// TwinCAT 3 PLC project PlcPrograme260424
// ProgramVersion: 3.1.4024.0
// libraries:
//   Tc2_EtherCAT, * (Beckhoff Automation GmbH)
//   Tc2_IoFunctions, * (Beckhoff Automation GmbH)
//   Tc2_MC2, * (Beckhoff Automation GmbH)
//   Tc2_ModbusRTU, * (Beckhoff Automation GmbH)
//   Tc2_NC, * (Beckhoff Automation GmbH)
//   Tc2_NcDrive, * (Beckhoff Automation GmbH)
//   Tc2_NCI, * (Beckhoff Automation GmbH)
//   Tc2_PlcInterpolation, * (Beckhoff Automation GmbH)
//   Tc2_SerialCom, * (Beckhoff Automation GmbH)
//   Tc2_Standard, * (Beckhoff Automation GmbH)
//   Tc2_SUPS, * (Beckhoff Automation GmbH)
//   Tc2_System, * (Beckhoff Automation GmbH)
//   Tc2_Utilities, * (Beckhoff Automation GmbH)
//   Tc3_MC2_AdvancedHoming, * (Beckhoff Automation GmbH)
//   Tc3_Module, * (Beckhoff Automation GmbH)
//   Util, * (System)
// project tree:
//   DUTs/Pump/ ST_Pump.TcDUT
//   DUTs/System/ ST_System.TcDUT
//   DUTs/气缸控制/ CylinderStatus.TcDUT, ST_YV.TcDUT
//   DUTs/真空控制/ ST_Vacuum.TcDUT
//   FB/01_Axis/DUTs/Axis_TouchProbeHome/ E_HomeStep.TcDUT, ST_HomeAdsGroup.TcDUT
//   FB/01_Axis/DUTs/Axis_DriveHome/ ST_HomeCoEGroup.TcDUT
//   FB/01_Axis/DUTs/ ST_Axis.TcDUT, ST_AxisControl.TcDUT, ST_AxisParameter.TcDUT, ST_AxisPosControl.TcDUT, ST_AxisPosPar.TcDUT, ST_AxisPosState.TcDUT, ST_AxisPos.TcDUT, ST_AxisState.TcDUT, ST_HomeViaDrivePar.TcDUT
//   FB/01_Axis/FB/ FB_Axis.TcPOU, FB_Axis_PE_Correct.TcPOU, FB_TouchProbe_Home_Bylimit.TcPOU, FB_Drive_Home.TcPOU
//   FB/02_NCI/FB/ FB_013_WriteZeroShiftEx.TcPOU, FB_010_ReadRParameter.TcPOU, FB_011WriteRParameter.TcPOU, FB_012_StepOnAfterStopEx.TcPOU, FB_01_NCI.TcPOU, FB_02_BuidGroup.TcPOU, FB_03_LoadProg.TcPOU, FB_04_Start.TcPOU, FB_05_ClearGrp.TcPOU, FB_06_ExSTOP.TcPOU, FB_07_FastMFunc.TcPOU, FB_08_ReSetEx.TcPOU, FB_09_SetOverridePercent.TcPOU
//   FB/05_YV/ FB_V_3B5.TcPOU
//   FB/06真空控制/ FB_VacuumControl.TcPOU
//   FB/11_AIO/DUTs/ ST_AIO.TcDUT
//   FB/11_AIO/FB/ FB_ADC.TcPOU, FB_DAC.TcPOU
//   FB/31_PDMSCtr/DUTs/ ST_LightCtr.TcDUT
//   FB/31_PDMSCtr/FB/ FB_PDMSCtr.TcPOU
//   FB/02_NCI/DUTs/ ST_IJP.TcDUT
//   FB/51_Netid/ FB_ReadNetid.TcPOU
//   FB/41_PosCom/DUTs/ ST_EL5131_CamCtrl.TcDUT
//   FB/41_PosCom/FB/ FB_013_POS_Comparition.TcPOU
//   FB/61_Alarm/DUTs/ Enum_ErrorClass.TcDUT, ST_Error.TcDUT, ST_HistoryError.TcDUT
//   FB/61_Alarm/FB/ FB_Alarm.TcPOU, FB_SetError.TcPOU, F_FormatWstringErrInfo.TcPOU
//   FB/71_Gear/DOUTs/ ST_Gear.TcDUT
//   FB/71_Gear/FB/ FB_Gear.TcPOU
//   GVLs/ Com_GVLS.TcGVL, GVL_ALM.TcGVL, GVL_IO.TcGVL, Programdata.TcGVL
//   / PlcTask.TcTTO
//   POUs/05_气缸控制/ YV_Ctrl.TcPOU
//   POUs/06_真空控制/ Vac_Ctrl.TcPOU
//   POUs/13_PosCompartion/ POS_Comparition.TcPOU
//   POUs/14_Bump/ Pump.TcPOU
//   POUs/15_Gear/ ProgGear.TcPOU
//   POUs/1_Axis/ AxisLink.TcPOU
//   POUs/2_Nci/ NCI_MAIN.TcPOU
//   POUs/3_Aio/ AIO.TcPOU
//   POUs/07_PDMctr/ PDMctr.TcPOU
//   POUs/ System_State.TcPOU
// real-time tasks:
//   TASK PlcTask: cycle T#1ms, priority 4, ADS port 350
// motion (NC):
//   TASK NC-Task 1 SAF: cycle T#1ms, priority 5, ADS port 501
//   TASK NC-Task 1 SVB: cycle T#2ms, priority 9, ADS port 511
//   AXIS X (id 1)
//     Dynamic: Acceleration=15000, Deceleration=15000, Jerk=150000
//     Velo: RefSync=1, SlowManual=10, FastManual=10, Fast=5
//     OtherSettings: AllowMotionCmdToSlave=true
//     encoder EncType=19
//       EncPara: ScaleFactorNumerator=1, ScaleFactorDenominator=10000, MaxCount=#xffffffff
//     drive DrvType=16
//       DrvPara: MaxCount=#xffffffff, DriveControlDWord=#x00020100
//         Analog: TorqueSetpointScale=10, ScaleFactorActTorque=0.1
//         TimeComp: TaskDelayCycles=1
//     controller CtrType=1
//       CtrPara: PriorControlFactor=1
//         Observer: BandWidth=20
//   AXIS Y (id 2)
//     Dynamic: Acceleration=15000, Deceleration=15000, Jerk=150000
//     Velo: RefSync=1, SlowManual=30, FastManual=30, Fast=5, Maximum=500
//     OtherSettings: AllowMotionCmdToSlave=true
//     encoder EncType=19
//       EncPara: ScaleFactorNumerator=1, ScaleFactorDenominator=10000, MaxCount=#xffffffff
//     drive DrvType=16
//       DrvPara: MaxCount=#xffffffff, DriveControlDWord=#x00020100
//         Analog: VeloReferenz=500, TorqueSetpointScale=10, ScaleFactorActTorque=0.1
//         TimeComp: TaskDelayCycles=1
//     controller CtrType=1
//       CtrPara: PriorControlFactor=1
//         Observer: BandWidth=20
//   AXIS R (id 3)
//     General: UnitName=°
//     Dynamic: AccelerationMaximum=50000, DecelerationMaximum=50000, Acceleration=50000, Deceleration=50000, Jerk=5000000
//     Velo: RefSync=1, SlowManual=5, FastManual=5, Fast=1000
//     OtherSettings: AllowMotionCmdToSlave=true
//     encoder EncType=19
//       EncPara: ScaleFactorNumerator=360, ScaleFactorDenominator=13107200, MaxCount=#xffffffff
//     drive DrvType=16
//       DrvPara: MaxCount=#xffffffff, DriveControlDWord=#x00020100
//         Analog: TorqueSetpointScale=10, ScaleFactorActTorque=0.1
//         TimeComp: TaskDelayCycles=1
//     controller CtrType=1
//       CtrPara: PriorControlFactor=1
//         Observer: BandWidth=20
//   AXIS Z1 (id 4)
//     Velo: RefSync=1, SlowManual=20, FastManual=20, Fast=200
//     OtherSettings: AllowMotionCmdToSlave=true
//     encoder EncType=19
//       EncPara: ScaleFactorNumerator=5, ScaleFactorDenominator=1048576, MaxCount=#xffffffff
//     drive DrvType=16
//       DrvPara: MaxCount=#xffffffff, DriveControlDWord=#x00000100
//         Analog: TorqueSetpointScale=10, ScaleFactorActTorque=0.1
//         TimeComp: TaskDelayCycles=1
//     controller CtrType=1
//       CtrPara: PriorControlFactor=1
//         Observer: BandWidth=20
//   AXIS Z2 (id 5)
//     Velo: RefSync=1, SlowManual=10, FastManual=10, Fast=200
//     OtherSettings: AllowMotionCmdToSlave=true
//     encoder EncType=19
//       EncPara: ScaleFactorNumerator=2, ScaleFactorDenominator=50000, Inverse=true, MaxCount=#xffffffff
//     drive DrvType=16
//       DrvPara: Inverse=true, MaxCount=#xffffffff, DriveControlDWord=#x00020000
//         Analog: TorqueSetpointScale=10, ScaleFactorActTorque=0.1
//         TimeComp: TaskDelayCycles=1
//     controller CtrType=1
//       CtrPara: PriorControlFactor=1
//         Observer: BandWidth=20
//   AXIS Pin (id 6)
//     Dynamic: AccelerationMaximum=5000, DecelerationMaximum=5000, Acceleration=5000, Deceleration=5000, Jerk=50000
//     Velo: SlowManual=3, FastManual=5, Maximum=5500
//     OtherSettings: AllowMotionCmdToSlave=true
//     encoder EncType=19
//       EncPara: ScaleFactorNumerator=360, ScaleFactorDenominator=10000, MaxCount=#xffffffff
//     drive DrvType=16
//       DrvPara: MaxCount=#xffffffff, DriveControlDWord=#x00020000
//         Analog: VeloReferenz=5000, TorqueSetpointScale=10, ScaleFactorActTorque=0.1
//         TimeComp: TaskDelayCycles=1
//     controller CtrType=1
//       CtrPara: PriorControlFactor=1
//         PosDiffControl: Range=50
//         Observer: BandWidth=20
//   AXIS R1 (id 7)
//     Velo: SlowManual=3, FastManual=5
//     OtherSettings: AllowMotionCmdToSlave=true
//     encoder EncType=19
//       EncPara: MaxCount=#xffffffff, ReferenceSystem=1
//     drive DrvType=16
//       DrvPara: MaxCount=#xffffffff, DriveControlDWord=#x00020000
//         Analog: TorqueSetpointScale=10, ScaleFactorActTorque=0.1
//         TimeComp: TaskDelayCycles=1
//     controller CtrType=1
//       CtrPara: PriorControlFactor=1
//         Observer: BandWidth=20
//   AXIS R2 (id 8)
//     Velo: SlowManual=3, FastManual=5
//     OtherSettings: AllowMotionCmdToSlave=true
//     encoder EncType=19
//       EncPara: MaxCount=#xffffffff, ReferenceSystem=1
//     drive DrvType=16
//       DrvPara: MaxCount=#xffffffff, DriveControlDWord=#x00020000
//         Analog: TorqueSetpointScale=10, ScaleFactorActTorque=0.1
//         TimeComp: TaskDelayCycles=1
//     controller CtrType=1
//       CtrPara: PriorControlFactor=1
//         Observer: BandWidth=20
//   AXIS R3 (id 9)
//     Velo: SlowManual=3, FastManual=5
//     OtherSettings: AllowMotionCmdToSlave=true
//     encoder EncType=19
//       EncPara: MaxCount=#xffffffff, ReferenceSystem=1
//     drive DrvType=16
//       DrvPara: MaxCount=#xffffffff, DriveControlDWord=#x00020000
//         Analog: TorqueSetpointScale=10, ScaleFactorActTorque=0.1
//         TimeComp: TaskDelayCycles=1
//     controller CtrType=1
//       CtrPara: PriorControlFactor=1
//         Observer: BandWidth=20
//   AXIS Bump (id 10)
//     Dynamic: Acceleration=100, Deceleration=100, Jerk=500
//     Velo: SlowManual=1, FastManual=3
//     TargetPosControl: Range=0.01
//     OtherSettings: AllowMotionCmdToSlave=true
//     encoder EncType=19
//       EncPara: ScaleFactorNumerator=0.01, ScaleFactorDenominator=10000, MaxCount=#xffffffff
//     drive DrvType=16
//       DrvPara: MaxCount=#xffffffff
//         Analog: TorqueSetpointScale=10, ScaleFactorActTorque=0.1
//         TimeComp: TaskDelayCycles=1
//     controller CtrType=1
//       CtrPara: PriorControlFactor=1
//         PosDiffControl: Enable=false, Range=20
//         Observer: BandWidth=20
// I/O:
//   DEVICE Device 1 (EtherCAT), AmsNetId 192.168.1.50.2.1
//     Term 1 (EK1200) [EK1200-5000 EtherCAT Power supply (2A E-Bus)]
//       Term 2 (EL1889) [EL1889 16Ch. Dig. Input 24V, 3ms, negative]
//       Term 3 (EL1889) [EL1889 16Ch. Dig. Input 24V, 3ms, negative]
//       Term 4 (EL2889) [EL2889 16Ch. Dig. Output 24V, 0.5A, negative]
//       Term 5 (EL3064) [EL3064 4Ch. Ana. Input 0-10V]
//       Term 6 (EL3064) [EL3064 4Ch. Ana. Input 0-10V]
//       Term 7 (EL4004) [EL4004 4Ch. Ana. Output 0-10V, 12bit]
//       Term 8 (EL4004) [EL4004 4Ch. Ana. Output 0-10V, 12bit]
//       Term 11 (EL6002) [EL6002 Interface 2Ch. (RS232)]
//       Term 12 (EK1110) [EK1110 EtherCAT extension]
//     Drive 13 (E2 CoE Drive) [E2 CoE Drive]
//     Drive 14 (E2 CoE Drive) [E2 CoE Drive]
//     Drive 15 (E2 CoE Drive) [E2 CoE Drive]
//     Drive 16 (SGDXS-xxxxA0x CoE Drive) [SGDXS-xxxxA0x EtherCAT(CoE) SERVOPACK Rev02.09]
//     Drive 17 (DM3C-EC522) [DM3C-EC522(COE)]
//     Drive 35 (AZD-KED) [AZD-KED rev0000]
//     Drive 37 (AZD4A-KED-1-3) [AZD4A-KED rev0301]
//     Drive 38 (AZD-KED) [AZD-KED rev0000]
// variable links:
//   NC-Task 1 SAF/Axes/Bump <-> Device 1 (EtherCAT)/Drive 38 (AZD-KED)
//     Drive/Inputs/In/nDcOutputTime <-> InfoData/DcOutputShift
//     Drive/Inputs/In/nState1 <-> Transmit PDO mapping 1/Statusword
//     Drive/Inputs/In/nState2 <-> Transmit PDO mapping 1/Statusword @bit 8
//     Drive/Inputs/In/nState4 @bit 1 <-> WcState/InputToggle
//     Drive/Inputs/In/nState4 <-> WcState/WcState
//     Drive/Inputs/In/nState5 <-> Transmit PDO mapping 1/Modes of operation display
//     Drive/Outputs/Out/nCtrl1 <-> Receive PDO mapping 1/Controlword
//     Drive/Outputs/Out/nCtrl2 <-> Receive PDO mapping 1/Controlword @bit 8
//     Drive/Outputs/Out/nCtrl5 <-> Receive PDO mapping 1/Modes of operation
//     Drive/Outputs/Out/nDataOut1 <-> Receive PDO mapping 1/Target position
//     Enc/Inputs/In/nDataIn1 <-> Transmit PDO mapping 1/Position actual value
//     Enc/Inputs/In/nDcInputTime <-> InfoData/DcInputShift
//     Enc/Inputs/In/nState4 @bit 1 <-> WcState/InputToggle
//     Enc/Inputs/In/nState4 <-> WcState/WcState
//   NC-Task 1 SAF/Axes/Pin <-> Device 1 (EtherCAT)/Drive 35 (AZD-KED)
//     Drive/Inputs/In/nDcOutputTime <-> InfoData/DcOutputShift
//     Drive/Inputs/In/nState1 <-> Transmit PDO mapping 1/Statusword
//     Drive/Inputs/In/nState2 <-> Transmit PDO mapping 1/Statusword @bit 8
//     Drive/Inputs/In/nState4 @bit 1 <-> WcState/InputToggle
//     Drive/Inputs/In/nState4 <-> WcState/WcState
//     Drive/Inputs/In/nState5 <-> Transmit PDO mapping 1/Modes of operation display
//     Drive/Outputs/Out/nCtrl1 <-> Receive PDO mapping 1/Controlword
//     Drive/Outputs/Out/nCtrl2 <-> Receive PDO mapping 1/Controlword @bit 8
//     Drive/Outputs/Out/nCtrl5 <-> Receive PDO mapping 1/Modes of operation
//     Drive/Outputs/Out/nDataOut1 <-> Receive PDO mapping 1/Target position
//     Enc/Inputs/In/nDataIn1 <-> Transmit PDO mapping 1/Position actual value
//     Enc/Inputs/In/nDcInputTime <-> InfoData/DcInputShift
//     Enc/Inputs/In/nState4 @bit 1 <-> WcState/InputToggle
//     Enc/Inputs/In/nState4 <-> WcState/WcState
//   NC-Task 1 SAF/Axes/R <-> Device 1 (EtherCAT)/Drive 15 (E2 CoE Drive)
//     Drive/Inputs/In/nDataIn1 <-> TxPDO 1/Following error actual value
//     Drive/Inputs/In/nDcOutputTime <-> InfoData/DcOutputShift
//     Drive/Inputs/In/nState1 <-> TxPDO 1/Statusword
//     Drive/Inputs/In/nState2 <-> TxPDO 1/Statusword @bit 8
//     Drive/Inputs/In/nState4 @bit 1 <-> WcState/InputToggle
//     Drive/Inputs/In/nState4 <-> WcState/WcState
//     Drive/Inputs/In/nState5 <-> TxPDO 1/Mode of operation display
//     Drive/Outputs/Out/nCtrl1 <-> RxPDO 1/Controlword
//     Drive/Outputs/Out/nCtrl2 <-> RxPDO 1/Controlword @bit 8
//     Drive/Outputs/Out/nCtrl5 <-> RxPDO 1/Mode of operation
//     Drive/Outputs/Out/nDataOut1 <-> RxPDO 1/Target Position
//     Enc/Inputs/In/nDataIn1 <-> TxPDO 1/Position actual value
//     Enc/Inputs/In/nDataIn3 <-> TxPDO 1/Touch Probe 1 positive edge
//     Enc/Inputs/In/nDcInputTime <-> InfoData/DcInputShift
//     Enc/Inputs/In/nState4 @bit 1 <-> WcState/InputToggle
//     Enc/Inputs/In/nState4 <-> WcState/WcState
//     Enc/Inputs/In/nState5 <-> TxPDO 1/Touch Probe status
//     Enc/Inputs/In/nState6 <-> TxPDO 1/Touch Probe status @bit 8
//     Enc/Outputs/Out/nCtrl5 <-> RxPDO 1/Touch probe function
//     Enc/Outputs/Out/nCtrl6 <-> RxPDO 1/Touch probe function @bit 8
//   NC-Task 1 SAF/Axes/R1 <-> Device 1 (EtherCAT)/Drive 37 (AZD4A-KED-1-3)
//     Drive/Inputs/In/nDcOutputTime <-> InfoData/DcOutputShift
//     Drive/Inputs/In/nState1 <-> Axis1 Transmit PDO mapping 1/Statusword
//     Drive/Inputs/In/nState2 <-> Axis1 Transmit PDO mapping 1/Statusword @bit 8
//     Drive/Inputs/In/nState4 @bit 1 <-> WcState/InputToggle
//     Drive/Inputs/In/nState4 <-> WcState/WcState
//     Drive/Inputs/In/nState5 <-> Axis1 Transmit PDO mapping 1/Modes of operation display
//     Drive/Outputs/Out/nCtrl1 <-> Axis1 Receive PDO mapping 1/Controlword
//     Drive/Outputs/Out/nCtrl2 <-> Axis1 Receive PDO mapping 1/Controlword @bit 8
//     Drive/Outputs/Out/nCtrl5 <-> Axis1 Receive PDO mapping 1/Modes of operation
//     Drive/Outputs/Out/nDataOut1 <-> Axis1 Receive PDO mapping 1/Target position
//     Enc/Inputs/In/nDataIn1 <-> Axis1 Transmit PDO mapping 1/Position actual value
//     Enc/Inputs/In/nDcInputTime <-> InfoData/DcInputShift
//     Enc/Inputs/In/nState4 @bit 1 <-> WcState/InputToggle
//     Enc/Inputs/In/nState4 <-> WcState/WcState
//   NC-Task 1 SAF/Axes/R2 <-> Device 1 (EtherCAT)/Drive 37 (AZD4A-KED-1-3)
//     Drive/Inputs/In/nDcOutputTime <-> InfoData/DcOutputShift
//     Drive/Inputs/In/nState1 <-> Axis2 Transmit PDO mapping 1/Statusword
//     Drive/Inputs/In/nState2 <-> Axis2 Transmit PDO mapping 1/Statusword @bit 8
//     Drive/Inputs/In/nState4 @bit 1 <-> WcState/InputToggle
//     Drive/Inputs/In/nState4 <-> WcState/WcState
//     Drive/Inputs/In/nState5 <-> Axis2 Transmit PDO mapping 1/Modes of operation display
//     Drive/Outputs/Out/nCtrl1 <-> Axis2 Receive PDO mapping 1/Controlword
//     Drive/Outputs/Out/nCtrl2 <-> Axis2 Receive PDO mapping 1/Controlword @bit 8
//     Drive/Outputs/Out/nCtrl5 <-> Axis2 Receive PDO mapping 1/Modes of operation
//     Drive/Outputs/Out/nDataOut1 <-> Axis2 Receive PDO mapping 1/Target position
//     Enc/Inputs/In/nDataIn1 <-> Axis2 Transmit PDO mapping 1/Position actual value
//     Enc/Inputs/In/nDcInputTime <-> InfoData/DcInputShift
//     Enc/Inputs/In/nState4 @bit 1 <-> WcState/InputToggle
//     Enc/Inputs/In/nState4 <-> WcState/WcState
//   NC-Task 1 SAF/Axes/R3 <-> Device 1 (EtherCAT)/Drive 37 (AZD4A-KED-1-3)
//     Drive/Inputs/In/nDcOutputTime <-> InfoData/DcOutputShift
//     Drive/Inputs/In/nState1 <-> Axis3 Transmit PDO mapping 1/Statusword
//     Drive/Inputs/In/nState2 <-> Axis3 Transmit PDO mapping 1/Statusword @bit 8
//     Drive/Inputs/In/nState4 @bit 1 <-> WcState/InputToggle
//     Drive/Inputs/In/nState4 <-> WcState/WcState
//     Drive/Inputs/In/nState5 <-> Axis3 Transmit PDO mapping 1/Modes of operation display
//     Drive/Outputs/Out/nCtrl1 <-> Axis3 Receive PDO mapping 1/Controlword
//     Drive/Outputs/Out/nCtrl2 <-> Axis3 Receive PDO mapping 1/Controlword @bit 8
//     Drive/Outputs/Out/nCtrl5 <-> Axis3 Receive PDO mapping 1/Modes of operation
//     Drive/Outputs/Out/nDataOut1 <-> Axis3 Receive PDO mapping 1/Target position
//     Enc/Inputs/In/nDataIn1 <-> Axis3 Transmit PDO mapping 1/Position actual value
//     Enc/Inputs/In/nDcInputTime <-> InfoData/DcInputShift
//     Enc/Inputs/In/nState4 @bit 1 <-> WcState/InputToggle
//     Enc/Inputs/In/nState4 <-> WcState/WcState
//   NC-Task 1 SAF/Axes/X <-> Device 1 (EtherCAT)/Drive 14 (E2 CoE Drive)
//     Drive/Inputs/In/nDataIn1 <-> TxPDO 1/Following error actual value
//     Drive/Inputs/In/nDcOutputTime <-> InfoData/DcOutputShift
//     Drive/Inputs/In/nState1 <-> TxPDO 1/Statusword
//     Drive/Inputs/In/nState2 <-> TxPDO 1/Statusword @bit 8
//     Drive/Inputs/In/nState4 @bit 1 <-> WcState/InputToggle
//     Drive/Inputs/In/nState4 <-> WcState/WcState
//     Drive/Inputs/In/nState5 <-> TxPDO 1/Mode of operation display
//     Drive/Outputs/Out/nCtrl1 <-> RxPDO 1/Controlword
//     Drive/Outputs/Out/nCtrl2 <-> RxPDO 1/Controlword @bit 8
//     Drive/Outputs/Out/nCtrl5 <-> RxPDO 1/Mode of operation
//     Drive/Outputs/Out/nDataOut1 <-> RxPDO 1/Target Position
//     Enc/Inputs/In/nDataIn1 <-> TxPDO 1/Position actual value
//     Enc/Inputs/In/nDataIn3 <-> TxPDO 1/Touch Probe 1 positive edge
//     Enc/Inputs/In/nDcInputTime <-> InfoData/DcInputShift
//     Enc/Inputs/In/nState4 @bit 1 <-> WcState/InputToggle
//     Enc/Inputs/In/nState4 <-> WcState/WcState
//     Enc/Inputs/In/nState5 <-> TxPDO 1/Touch Probe status
//     Enc/Inputs/In/nState6 <-> TxPDO 1/Touch Probe status @bit 8
//     Enc/Outputs/Out/nCtrl5 <-> RxPDO 1/Touch probe function
//     Enc/Outputs/Out/nCtrl6 <-> RxPDO 1/Touch probe function @bit 8
//   NC-Task 1 SAF/Axes/Y <-> Device 1 (EtherCAT)/Drive 13 (E2 CoE Drive)
//     Drive/Inputs/In/nDataIn1 <-> TxPDO 1/Following error actual value
//     Drive/Inputs/In/nDcOutputTime <-> InfoData/DcOutputShift
//     Drive/Inputs/In/nState1 <-> TxPDO 1/Statusword
//     Drive/Inputs/In/nState2 <-> TxPDO 1/Statusword @bit 8
//     Drive/Inputs/In/nState4 @bit 1 <-> WcState/InputToggle
//     Drive/Inputs/In/nState4 <-> WcState/WcState
//     Drive/Inputs/In/nState5 <-> TxPDO 1/Mode of operation display
//     Drive/Outputs/Out/nCtrl1 <-> RxPDO 1/Controlword
//     Drive/Outputs/Out/nCtrl2 <-> RxPDO 1/Controlword @bit 8
//     Drive/Outputs/Out/nCtrl5 <-> RxPDO 1/Mode of operation
//     Drive/Outputs/Out/nDataOut1 <-> RxPDO 1/Target Position
//     Enc/Inputs/In/nDataIn1 <-> TxPDO 1/Position actual value
//     Enc/Inputs/In/nDataIn3 <-> TxPDO 1/Touch Probe 1 positive edge
//     Enc/Inputs/In/nDcInputTime <-> InfoData/DcInputShift
//     Enc/Inputs/In/nState4 @bit 1 <-> WcState/InputToggle
//     Enc/Inputs/In/nState4 <-> WcState/WcState
//     Enc/Inputs/In/nState5 <-> TxPDO 1/Touch Probe status
//     Enc/Inputs/In/nState6 <-> TxPDO 1/Touch Probe status @bit 8
//     Enc/Outputs/Out/nCtrl5 <-> RxPDO 1/Touch probe function
//     Enc/Outputs/Out/nCtrl6 <-> RxPDO 1/Touch probe function @bit 8
//   NC-Task 1 SAF/Axes/Z1 <-> Device 1 (EtherCAT)/Drive 16 (SGDXS-xxxxA0x CoE Drive)
//     Drive/Inputs/In/nDataIn1 <-> 1st Transmit PDO mapping/Following error actual value
//     Drive/Inputs/In/nDataIn3[0] <-> 1st Transmit PDO mapping/Torque actual value
//     Drive/Inputs/In/nDcOutputTime <-> InfoData/DcOutputShift
//     Drive/Inputs/In/nState1 <-> 1st Transmit PDO mapping/Status word
//     Drive/Inputs/In/nState2 <-> 1st Transmit PDO mapping/Status word @bit 8
//     Drive/Inputs/In/nState4 @bit 1 <-> WcState/InputToggle
//     Drive/Inputs/In/nState4 <-> WcState/WcState
//     Drive/Inputs/In/nState5 <-> 1st Transmit PDO mapping/Modes of operation display
//     Drive/Outputs/Out/nCtrl1 <-> 1st Receive PDO mapping/Control word
//     Drive/Outputs/Out/nCtrl2 <-> 1st Receive PDO mapping/Control word @bit 8
//     Drive/Outputs/Out/nCtrl5 <-> 1st Receive PDO mapping/Modes of operation
//     Drive/Outputs/Out/nDataOut1 <-> 1st Receive PDO mapping/Target position
//     Drive/Outputs/Out/nDataOut2 <-> 1st Receive PDO mapping/Target velocity
//     Drive/Outputs/Out/nDataOut4[0] <-> 1st Receive PDO mapping/Target torque
//     Enc/Inputs/In/nDataIn1 <-> 1st Transmit PDO mapping/Position actual value
//     Enc/Inputs/In/nDataIn3 <-> 1st Transmit PDO mapping/Touch probe 1 position value
//     Enc/Inputs/In/nDcInputTime <-> InfoData/DcInputShift
//     Enc/Inputs/In/nState4 @bit 1 <-> WcState/InputToggle
//     Enc/Inputs/In/nState4 <-> WcState/WcState
//     Enc/Inputs/In/nState5 <-> 1st Transmit PDO mapping/Touch probe status
//     Enc/Inputs/In/nState6 <-> 1st Transmit PDO mapping/Touch probe status @bit 8
//     Enc/Outputs/Out/nCtrl5 <-> 1st Receive PDO mapping/Touch probe function
//     Enc/Outputs/Out/nCtrl6 <-> 1st Receive PDO mapping/Touch probe function @bit 8
//   NC-Task 1 SAF/Axes/Z2 <-> Device 1 (EtherCAT)/Drive 17 (DM3C-EC522)
//     Drive/Inputs/In/nDcOutputTime <-> InfoData/DcOutputShift
//     Drive/Inputs/In/nState1 <-> Transmit PDO 1/Status Word
//     Drive/Inputs/In/nState2 <-> Transmit PDO 1/Status Word @bit 8
//     Drive/Inputs/In/nState4 @bit 1 <-> WcState/InputToggle
//     Drive/Inputs/In/nState4 <-> WcState/WcState
//     Drive/Outputs/Out/nCtrl1 <-> Receive PDO 1/Control Word
//     Drive/Outputs/Out/nCtrl2 <-> Receive PDO 1/Control Word @bit 8
//     Drive/Outputs/Out/nDataOut1 <-> Receive PDO 1/Profile Target Position
//     Enc/Inputs/In/nDataIn1 <-> Transmit PDO 1/Position Actual Value
//     Enc/Inputs/In/nDataIn3 <-> Transmit PDO 1/Touch Probe 1 Positive Value
//     Enc/Inputs/In/nDcInputTime <-> InfoData/DcInputShift
//     Enc/Inputs/In/nState4 @bit 1 <-> WcState/InputToggle
//     Enc/Inputs/In/nState4 <-> WcState/WcState
//     Enc/Inputs/In/nState5 <-> Transmit PDO 1/Touch Probe Status
//     Enc/Inputs/In/nState6 <-> Transmit PDO 1/Touch Probe Status @bit 8
//     Enc/Outputs/Out/nCtrl5 <-> Receive PDO 1/Touch Probe Function
//     Enc/Outputs/Out/nCtrl6 <-> Receive PDO 1/Touch Probe Function @bit 8
//   PlcPrograme260424/PlcPrograme260424 Instance <-> Device 1 (EtherCAT)
//     PlcTask Inputs/System_State.fbReadNetid.tAmsNetid <-> InfoData/AmsNetId
//   PlcPrograme260424/PlcPrograme260424 Instance <-> Device 1 (EtherCAT)/Drive 13 (E2 CoE Drive)
//     PlcTask Inputs/Com_GVLS.arstAxis[1].uiSlaveAddr <-> InfoData/AdsAddr/port
//   PlcPrograme260424/PlcPrograme260424 Instance <-> Device 1 (EtherCAT)/Drive 14 (E2 CoE Drive)
//     PlcTask Inputs/Com_GVLS.arstAxis[2].uiSlaveAddr <-> InfoData/AdsAddr/port
//   PlcPrograme260424/PlcPrograme260424 Instance <-> Device 1 (EtherCAT)/Drive 15 (E2 CoE Drive)
//     PlcTask Inputs/Com_GVLS.arstAxis[3].uiSlaveAddr <-> InfoData/AdsAddr/port
//   PlcPrograme260424/PlcPrograme260424 Instance <-> Device 1 (EtherCAT)/Drive 16 (SGDXS-xxxxA0x CoE Drive)
//     PlcTask Inputs/Com_GVLS.arstAxis[4].uiSlaveAddr <-> InfoData/AdsAddr/port
//   PlcPrograme260424/PlcPrograme260424 Instance <-> Device 1 (EtherCAT)/Drive 17 (DM3C-EC522)
//     PlcTask Inputs/Com_GVLS.arstAxis[5].uiSlaveAddr <-> InfoData/AdsAddr/port
//   PlcPrograme260424/PlcPrograme260424 Instance <-> Device 1 (EtherCAT)/Drive 35 (AZD-KED)
//     PlcTask Inputs/Com_GVLS.arstAxis[6].uiSlaveAddr <-> InfoData/AdsAddr/port
//   PlcPrograme260424/PlcPrograme260424 Instance <-> Device 1 (EtherCAT)/Drive 37 (AZD4A-KED-1-3)
//     PlcTask Inputs/Com_GVLS.arstAxis[7].uiSlaveAddr <-> InfoData/AdsAddr/port
//     PlcTask Inputs/Com_GVLS.arstAxis[8].uiSlaveAddr <-> InfoData/AdsAddr/port
//     PlcTask Inputs/Com_GVLS.arstAxis[9].uiSlaveAddr <-> InfoData/AdsAddr/port
//   PlcPrograme260424/PlcPrograme260424 Instance <-> Device 1 (EtherCAT)/Drive 38 (AZD-KED)
//     PlcTask Inputs/Com_GVLS.arstAxis[10].uiSlaveAddr <-> InfoData/AdsAddr/port
//   PlcPrograme260424/PlcPrograme260424 Instance <-> Device 1 (EtherCAT)/Term 1 (EK1200)/Term 11 (EL6002)
//     PlcTask Inputs/PDMctr.FB_PDMSCtr.COMin_MASTER @bit {16..184 step 8} <-> COM TxPDO-Map Inputs Channel 1/Data In {0..21}  (22 links)
//     PlcTask Inputs/PDMctr.FB_PDMSCtr.COMin_MASTER <-> COM TxPDO-Map Inputs Channel 1/Status
//     PlcTask Outputs/PDMctr.FB_PDMSCtr.COMout_MASTER <-> COM RxPDO-Map Outputs Channel 1/Ctrl
//     PlcTask Outputs/PDMctr.FB_PDMSCtr.COMout_MASTER @bit {16..184 step 8} <-> COM RxPDO-Map Outputs Channel 1/Data Out {0..21}  (22 links)
//   PlcPrograme260424/PlcPrograme260424 Instance <-> Device 1 (EtherCAT)/Term 1 (EK1200)/Term 2 (EL1889)
//     PlcTask Inputs/GVL_IO.X000001 <-> Channel 1/Input
//     PlcTask Inputs/GVL_IO.X000002 <-> Channel 2/Input
//     PlcTask Inputs/GVL_IO.X000003 <-> Channel 3/Input
//     PlcTask Inputs/GVL_IO.X000004 <-> Channel 4/Input
//     PlcTask Inputs/GVL_IO.X000005 <-> Channel 5/Input
//     PlcTask Inputs/GVL_IO.X000006 <-> Channel 6/Input
//     PlcTask Inputs/GVL_IO.X000007 <-> Channel 7/Input
//     PlcTask Inputs/GVL_IO.X000008 <-> Channel 8/Input
//     PlcTask Inputs/GVL_IO.X000009 <-> Channel 9/Input
//     PlcTask Inputs/GVL_IO.X000010 <-> Channel 10/Input
//     PlcTask Inputs/GVL_IO.X000011 <-> Channel 11/Input
//     PlcTask Inputs/GVL_IO.X000012 <-> Channel 12/Input
//     PlcTask Inputs/GVL_IO.X000013 <-> Channel 13/Input
//     PlcTask Inputs/GVL_IO.X000014 <-> Channel 14/Input
//     PlcTask Inputs/GVL_IO.X000015 <-> Channel 15/Input
//     PlcTask Inputs/GVL_IO.X000016 <-> Channel 16/Input
//   PlcPrograme260424/PlcPrograme260424 Instance <-> Device 1 (EtherCAT)/Term 1 (EK1200)/Term 3 (EL1889)
//     PlcTask Inputs/GVL_IO.X001001 <-> Channel 1/Input
//     PlcTask Inputs/GVL_IO.X001002 <-> Channel 2/Input
//     PlcTask Inputs/GVL_IO.X001003 <-> Channel 3/Input
//     PlcTask Inputs/GVL_IO.X001004 <-> Channel 4/Input
//     PlcTask Inputs/GVL_IO.X001005 <-> Channel 5/Input
//     PlcTask Inputs/GVL_IO.X001006 <-> Channel 6/Input
//     PlcTask Inputs/GVL_IO.X001007 <-> Channel 7/Input
//     PlcTask Inputs/GVL_IO.X001008 <-> Channel 8/Input
//     PlcTask Inputs/GVL_IO.X001009 <-> Channel 9/Input
//     PlcTask Inputs/GVL_IO.X001010 <-> Channel 10/Input
//     PlcTask Inputs/GVL_IO.X001011 <-> Channel 11/Input
//     PlcTask Inputs/GVL_IO.X001012 <-> Channel 12/Input
//     PlcTask Inputs/GVL_IO.X001013 <-> Channel 13/Input
//     PlcTask Inputs/GVL_IO.X001014 <-> Channel 14/Input
//     PlcTask Inputs/GVL_IO.X001015 <-> Channel 15/Input
//     PlcTask Inputs/GVL_IO.X001016 <-> Channel 16/Input
//   PlcPrograme260424/PlcPrograme260424 Instance <-> Device 1 (EtherCAT)/Term 1 (EK1200)/Term 4 (EL2889)
//     PlcTask Outputs/GVL_IO.Y000001 <-> Channel 1/Output
//     PlcTask Outputs/GVL_IO.Y000002 <-> Channel 2/Output
//     PlcTask Outputs/GVL_IO.Y000003 <-> Channel 3/Output
//     PlcTask Outputs/GVL_IO.Y000004 <-> Channel 4/Output
//     PlcTask Outputs/GVL_IO.Y000005 <-> Channel 5/Output
//     PlcTask Outputs/GVL_IO.Y000006 <-> Channel 6/Output
//     PlcTask Outputs/GVL_IO.Y000007 <-> Channel 7/Output
//     PlcTask Outputs/GVL_IO.Y000008 <-> Channel 8/Output
//     PlcTask Outputs/GVL_IO.Y000009 <-> Channel 9/Output
//     PlcTask Outputs/GVL_IO.Y000010 <-> Channel 10/Output
//     PlcTask Outputs/GVL_IO.Y000011 <-> Channel 11/Output
//     PlcTask Outputs/GVL_IO.Y000012 <-> Channel 12/Output
//     PlcTask Outputs/GVL_IO.Y000013 <-> Channel 13/Output
//     PlcTask Outputs/GVL_IO.Y000014 <-> Channel 14/Output
//     PlcTask Outputs/GVL_IO.Y000015 <-> Channel 15/Output
//     PlcTask Outputs/GVL_IO.Y000016 <-> Channel 16/Output
//   PlcPrograme260424/PlcPrograme260424 Instance <-> Device 1 (EtherCAT)/Term 1 (EK1200)/Term 5 (EL3064)
//     PlcTask Inputs/Programdata.AX_1[{1..4}] <-> AI Standard Channel {1..4}/Value  (4 links)
//   PlcPrograme260424/PlcPrograme260424 Instance <-> Device 1 (EtherCAT)/Term 1 (EK1200)/Term 6 (EL3064)
//     PlcTask Inputs/Programdata.AX_2[{1..4}] <-> AI Standard Channel {1..4}/Value  (4 links)
//   PlcPrograme260424/PlcPrograme260424 Instance <-> Device 1 (EtherCAT)/Term 1 (EK1200)/Term 7 (EL4004)
//     PlcTask Outputs/Programdata.AY_1[{1..4}] <-> AO Outputs Channel {1..4}/Analog output  (4 links)
//   PlcPrograme260424/PlcPrograme260424 Instance <-> Device 1 (EtherCAT)/Term 1 (EK1200)/Term 8 (EL4004)
//     PlcTask Outputs/Programdata.AY_2[{1..4}] <-> AO Outputs Channel {1..4}/Analog output  (4 links)
//   PlcPrograme260424/PlcPrograme260424 Instance <-> NC-Task 1 SAF/Axes/Bump
//     PlcTask Inputs/Programdata.arAXIS[10].NcToPlc <-> Outputs/ToPlc
//     PlcTask Outputs/Programdata.arAXIS[10].PlcToNc <-> Inputs/FromPlc
//   PlcPrograme260424/PlcPrograme260424 Instance <-> NC-Task 1 SAF/Axes/Pin
//     PlcTask Inputs/Programdata.arAXIS[6].NcToPlc <-> Outputs/ToPlc
//     PlcTask Outputs/Programdata.arAXIS[6].PlcToNc <-> Inputs/FromPlc
//   PlcPrograme260424/PlcPrograme260424 Instance <-> NC-Task 1 SAF/Axes/R
//     PlcTask Inputs/Programdata.arAXIS[3].NcToPlc <-> Outputs/ToPlc
//     PlcTask Outputs/Programdata.arAXIS[3].PlcToNc <-> Inputs/FromPlc
//   PlcPrograme260424/PlcPrograme260424 Instance <-> NC-Task 1 SAF/Axes/R1
//     PlcTask Inputs/Programdata.arAXIS[7].NcToPlc <-> Outputs/ToPlc
//     PlcTask Outputs/Programdata.arAXIS[7].PlcToNc <-> Inputs/FromPlc
//   PlcPrograme260424/PlcPrograme260424 Instance <-> NC-Task 1 SAF/Axes/R2
//     PlcTask Inputs/Programdata.arAXIS[8].NcToPlc <-> Outputs/ToPlc
//     PlcTask Outputs/Programdata.arAXIS[8].PlcToNc <-> Inputs/FromPlc
//   PlcPrograme260424/PlcPrograme260424 Instance <-> NC-Task 1 SAF/Axes/R3
//     PlcTask Inputs/Programdata.arAXIS[9].NcToPlc <-> Outputs/ToPlc
//     PlcTask Outputs/Programdata.arAXIS[9].PlcToNc <-> Inputs/FromPlc
//   PlcPrograme260424/PlcPrograme260424 Instance <-> NC-Task 1 SAF/Axes/X
//     PlcTask Inputs/Programdata.arAXIS[1].NcToPlc <-> Outputs/ToPlc
//     PlcTask Outputs/Programdata.arAXIS[1].PlcToNc <-> Inputs/FromPlc
//   PlcPrograme260424/PlcPrograme260424 Instance <-> NC-Task 1 SAF/Axes/Y
//     PlcTask Inputs/Programdata.arAXIS[2].NcToPlc <-> Outputs/ToPlc
//     PlcTask Outputs/Programdata.arAXIS[2].PlcToNc <-> Inputs/FromPlc
//   PlcPrograme260424/PlcPrograme260424 Instance <-> NC-Task 1 SAF/Axes/Z1
//     PlcTask Inputs/Programdata.arAXIS[4].NcToPlc <-> Outputs/ToPlc
//     PlcTask Outputs/Programdata.arAXIS[4].PlcToNc <-> Inputs/FromPlc
//   PlcPrograme260424/PlcPrograme260424 Instance <-> NC-Task 1 SAF/Axes/Z2
//     PlcTask Inputs/Programdata.arAXIS[5].NcToPlc <-> Outputs/ToPlc
//     PlcTask Outputs/Programdata.arAXIS[5].PlcToNc <-> Inputs/FromPlc
//   PlcPrograme260424/PlcPrograme260424 Instance <-> NC-Task 1 SAF/Channel 2
//     PlcTask Inputs/Com_GVLS.stIJP.in_stItpToPlc <-> Outputs/ToPlc
//     PlcTask Outputs/Com_GVLS.stIJP.out_stItpToPlc <-> Inputs/FromPlc

CONFIGURATION PlcPrograme260424
    RESOURCE PLC ON TwinCAT3
        TASK PlcTask(INTERVAL := T#1ms, PRIORITY := 4);
        PROGRAM AxisLink WITH PlcTask : AxisLink;
        PROGRAM NCI_MAIN WITH PlcTask : NCI_MAIN;
        PROGRAM AIO WITH PlcTask : AIO;
        PROGRAM System_State WITH PlcTask : System_State;
        PROGRAM PDMctr WITH PlcTask : PDMctr;
        PROGRAM Vac_Ctrl WITH PlcTask : Vac_Ctrl;
        PROGRAM POS_Comparition WITH PlcTask : POS_Comparition;
        PROGRAM ProgGear WITH PlcTask : ProgGear;
        PROGRAM YV_Ctrl WITH PlcTask : YV_Ctrl;
        PROGRAM Pump WITH PlcTask : Pump;
    END_RESOURCE
END_CONFIGURATION

// ---- DUTs/Pump/ST_Pump.TcDUT
TYPE ST_Pump :
STRUCT
	rJogVel_A								:REAL				    ;			// 流速	
	rJogVol_A								:REAL				    ;			// 容积
	strml               :STRING:='5ml'               ;  //当前进样器容积
	rInjectDia          :ARRAY[1..2] OF REAL  :=[ 7.3, 10.3]; //当前进样器内径
	rVol_Process1   : REAL;  // 流程1：快速注入容量 (ul)
    rVel_Process1   : REAL;  // 流程1：快速注入流速 (ul/min)
    rVel_Process2   : REAL;  // 流程2：匀速注入流速 (ul/min)
    rVol_Process3   : REAL;  // 流程3：快速抽取容量 (ul)
    rVel_Process3   : REAL;  // 流程3：快速抽取流速 (ul/min)
	iCurrentStep    : INT;    // 当前运行状态 (0:待机, 10:注入准备, 11:快速注入中..., 20:匀速注入中..., 30:抽取中..., 31:抽取中...)
	bEX_PumpTrigOn  : BOOL;   //注射泵触发开
	bEX_PumpTrigOff  : BOOL;   //注射泵触发关

END_STRUCT
END_TYPE

// ---- DUTs/System/ST_System.TcDUT
TYPE ST_System :
STRUCT
	    strNetID                                                               :STRING;
        bSystemPowerOn                                        :BOOL                                                        ;                        //系统动力电上电标志        
        bManual                                                        :BOOL                                                        ;                        //手自动标志
        bReset                                                        :BOOL                                                        ;                        //复位
        bStop                                                        :BOOL                                                        ;                        //停止
        bEMG                                                               :BOOL                                                        ;                        //急停
        bSafetyDoor                                                :BOOL                                                        ;                        //安全门
        bLightOn                                                :BOOL                                                        ;                        //照明灯
        bAxesPowerOK                                            :BOOL                                                        ;                        //所有轴均上使能
        bAxesHomeOK                                                :BOOL                                                        ;                        //所有轴均回零完成
	bHOME                             :BOOL                                      ;           // 整机回零
	bHoming                           :BOOL                                      ;           // 整机回零中
	bHOMEOK                           :BOOL                                      ;           // 整机回零完成
	bPower                            :BOOL                                      ;           // 整机使能
	bPowerOK                          :BOOL                                      ;           // 整机使能完成
	bUVon                             :BOOL                                      ;           // UV开关
	bUVErr                            :BOOL                                      ;           // UV开关报错
        bAxesInMotion                                        :BOOL                                                        ;                        //有轴移动
        bError                                                        :BOOL                                                        ;                        //报错
        bWarning                                                :BOOL                                                        ;                        //警告
        bLightError                                                :BOOL                                                        ;                        //轻量错误
        bCriticalError                                        :BOOL                                                        ;                        //严重错误
        bErrorUpdate                                        :BOOL                                                           ;                        //出现新的报错                                        
        arErrorID                                                :ARRAY[0..999] OF BOOL                                     ;                        //报警索引号
        arstrErrorInfo                                        :ARRAY[0..999] OF STRING                                      ;                        //报警信息（英）
        strDeviceName                                        :STRING                                                        ;                        //设备名称
        uiPinNum                                                :UINT                                                        ;                        //剥离头类型，1-单电机，2-双电机
	    bSignalLampRed	                                       :BOOL	; // 三色灯-红                   
        bSignalLampGreen	                                    :BOOL	 ;// 三色灯-绿
        bSignalLampYellow	                                     :BOOL	 ;// 三色灯-黄
        bSingalLampBuzzle	                                      :BOOL	; // 三色灯-蜂鸣器
END_STRUCT
END_TYPE

// ---- DUTs/气缸控制/CylinderStatus.TcDUT
(* 单个气缸状态 *)
TYPE CylinderStatus :
STRUCT
    bExtendReq    : BOOL;   // 伸出请求
    bRetractReq   : BOOL;   // 回缩请求
    q_bExtend     : BOOL;   // 输出伸出
    q_bRetract    : BOOL;   // 输出回缩
    xExtendPos    : BOOL;   // 伸出到位
    xRetractPos   : BOOL;   // 回缩到位
    bInDeadtime   : BOOL;   // 死区标志
    bAlarm        : BOOL;   // 报警状态
END_STRUCT
END_TYPE

// ---- DUTs/气缸控制/ST_YV.TcDUT
TYPE ST_YV :
STRUCT
	bYVFw_A   :BOOL; //  伸出操作
	bYVBw_A   :BOOL; //  缩回操作
	bYVFw_In  :BOOL; //  伸出限位
	bYVBw_In  :BOOL; //  缩回限位
	bYVFw_OK  :BOOL; //  气缸伸出到位
	bYVBw_OK  :BOOL; //  气缸缩回到位
	bYVFw_Out :BOOL; //  硬件输出
	bYVBw_Out :BOOL; //  硬件输出
	bError	  :BOOL; //  错误状态
	//arErrorID :UINT; //  错误ID
	udiError  :UDINT; //  错误ID
	arErrorID	  :ARRAY[0..7] OF BOOL   ;   // 错误ID,上位机需求

END_STRUCT
END_TYPE

// ---- DUTs/真空控制/ST_Vacuum.TcDUT
(*

TYPE ST_Vacuum :
STRUCT
    (* 输入 *)
    bVacuumReq     : BOOL;   // 抽真空请求
    bReleaseReq    : BOOL;   // 破真空请求
    xVacuumOk      : BOOL;   // 真空到位信号

    (* 输出 *)
    qVacuumValve   : BOOL;   // 真空阀
    qReleaseValve  : BOOL;   // 破真空阀

    (* 状态 *)
    bVacuumDone    : BOOL;
    bAlarm         : BOOL;
END_STRUCT
END_TYPE

*)

TYPE ST_Vacuum :
STRUCT
    (* 输入 *)
    bVacuumReq      : BOOL;   // 抽真空请求
END_STRUCT
END_TYPE

// ---- FB/01_Axis/DUTs/Axis_TouchProbeHome/E_HomeStep.TcDUT
//{attribute 'qualified_only'}
{attribute 'strict'}
TYPE E_HomeStep :
(
	IndexHomeInital:=0,
	AckHomeDirection,
	SetParameter,
	SetParameterState,
	ReadParameter,
	ReadParameterState,
	AckParameter,
	ExecuteToOrigin,
	HomeMonitorState,
	HomeMoveABS,
	ExecuteHomeDone,
	IndexHomeErrorState
);
END_TYPE

// ---- FB/01_Axis/DUTs/Axis_TouchProbeHome/ST_HomeAdsGroup.TcDUT
TYPE ST_HomeAdsGroup :
STRUCT
    nCalibrationVel			:UDINT:=16#4001;				(* 回零速度ADS地址*)	
	nHomeInfo				:UDINT:=16#5001;				(* 回零参数ADS地址*)

END_STRUCT
END_TYPE

// ---- FB/01_Axis/DUTs/Axis_DriveHome/ST_HomeCoEGroup.TcDUT
TYPE ST_HomeCoEGroup :
STRUCT
	strNetID			    :STRING:='192.168.1.50.2.1';				(* 回零速度coe地址*)	
	wSlaveAddr				:WORD:=1001;				                (* 回零参数coe地址*)
	uiAxisChannelNum        :WORD:=1;                                   (* 一拖多驱动器COE地址递增index*)
END_STRUCT
END_TYPE

// ---- FB/01_Axis/DUTs/ST_Axis.TcDUT
TYPE ST_Axis :
STRUCT
	strName			:STRING					    ;
	wstrName		:WSTRING				    ;
	strNetID        :STRING;
	uiSlaveAddr     AT%I*  :WORD;
	Control			:ST_AxisControl				;		
	Parameter		:ST_AxisParameter			;		
	State			:ST_AxisState				;	
	Pos				:ST_AxisPos		            ;
END_STRUCT
END_TYPE

// ---- FB/01_Axis/DUTs/ST_AxisControl.TcDUT

TYPE ST_AxisControl :
STRUCT
	bPowerOn			:BOOL				;		//伺服使能	
	bHome_M				:BOOL				;		//手动回零	
	bHome_A				:BOOL				;		//自动回零	
	bHome_Con			:BOOL				;		//回零条件	
	bJogCw_M			:BOOL				;		//手动点动加（顺时针）	
	bJogCcw_M			:BOOL				;		//手动点动减（逆时针）	
	bJogCw_A			:BOOL				;		//自动点动加（顺时针）	
	bJogCcw_A			:BOOL				;		//自动点动减（逆时针）		
	bJogCw_Con			:BOOL				;		//点动加条件	
	bJogCcw_Con			:BOOL				;		//点动减条件	
	bStop_A				:BOOL				;		//自动停止	
	bStop_M				:BOOL				;		//手动停止	
	bSetPos				:BOOL				;		//置位	
	iJogMode			:INT				;		//Jog运行模式0-连续 1-点动
	bReset_A			:BOOL				;
	bReset_M			:BOOL				;
END_STRUCT
END_TYPE

// ---- FB/01_Axis/DUTs/ST_AxisParameter.TcDUT
TYPE ST_AxisParameter :
STRUCT	
	rMaxVel									:REAL				;			//额定最大速度	
	rHmOffset								:REAL				;			//原点偏差值(单原点回零时使用)	
	rHmVel									:REAL				;			//回零速度	
	rHmAcc									:REAL				;			//回零加速度	
	rHmDec									:REAL				;			//回零减速度	
	rHmJerk									:REAL				;			//回零跃度	
	rJogVel_M								:REAL				;			//手动点动速度	
	rJogAcc_M								:REAL				;			//手动点动加速度	
	rJogDec_M								:REAL				;			//手动点动减速度
	rJogPos_M								:REAL				;			//手动寸动增量	
	rJogVel_A								:REAL				;			//自动点动速度	
	rJogAcc_A								:REAL				;			//自动点动加速度	
	rJogDec_A								:REAL				;			//自动点动减速度	
	rJogPos_A								:REAL				;			//自动寸动增量	
	rStopDec								:REAL				;			//停止减速度	
	rStopJerk								:REAL				;			//停止跃度	
	rSetPos									:REAL				;			//置位位置	
	udiPDO_60FD				AT%I*			:UDINT				;			//限位原点接入驱动器下配置：数字输入
	udiPDO_6071				AT%Q*			:INT				;			// 输入力矩
//	uiPDO_60B8				AT%Q*			:UINT				;			//探针回零模式下配置：探针控制字
//	uiPDO_60B9				AT%I*			:UINT				;			//探针回零模式下配置：探针状态字	
	uiHomeMode								:UINT				;			//0=碰限位回零 , 1=单原点回零 , 2=限位+原点光电回零,6=驱动器回零,8=模块限位+驱动器回零	
	iTorque									:INT				;			//设定转矩
	bAbsEnc									:BOOL				;			//true= 绝对值编码器，false= 增量式编码器	
	bHmDir									:BOOL				;			//FALSE=正向回零 , TRUE=反向回零	
//	diPDO_60BA		 		AT%I*			:DINT				;			//探针回零模式下配置：探针1上升沿	
	diPDO_6064								:DINT				;			//轴当前脉冲数
	rInPosValue                     		:REAL	:=0.01		;			// 运动到位
	rSetPosition							:REAL				;			// 回退距离
	uiAxisChannelNum						:UINT	:=1			;			//针对多轴驱动器中的轴通道号,单轴按通道1计算
	rTorque                                 :REAL               ;           // 力矩模式设定力矩6071
	sthomeViaDrivePar 				:ST_HomeViaDrivePar			;			
END_STRUCT
END_TYPE

// ---- FB/01_Axis/DUTs/ST_AxisPosControl.TcDUT
TYPE ST_AxisPosControl :
STRUCT
	bGo_Con			:			BOOL			;		//定位条件
	bGo_M			:			BOOL			;		//手动定位启动
	bGo_A			:			BOOL			;		//自动定位启动
END_STRUCT
END_TYPE

// ---- FB/01_Axis/DUTs/ST_AxisPosPar.TcDUT
TYPE ST_AxisPosPar :
STRUCT
	bRelEnable			:BOOL		;		//FALSE绝对定位，TRUE相对定位	
	rPos				:REAL		;		//定位位置	
	rVel				:REAL		;		//定位速度	
	rAcc				:REAL		;		//定位加速度	
	rDec				:REAL		;		//定位减速度	
	rJerk				:REAL		;		//定位跃度	
END_STRUCT
END_TYPE

// ---- FB/01_Axis/DUTs/ST_AxisPosState.TcDUT
TYPE ST_AxisPosState :
STRUCT
	bGo_OK			:BOOL		;		//定位完成	
	bGo_Moving		:BOOL		;		//定位中	
	rGo_CT			:REAL		;		//定位持续时间	
END_STRUCT
END_TYPE

// ---- FB/01_Axis/DUTs/ST_AxisPos.TcDUT
TYPE ST_AxisPos :
STRUCT
	Ctrl			:			ST_AxisPosControl	;
	Par				:			ST_AxisPosPar		;
	State			:			ST_AxisPosState		;
END_STRUCT
END_TYPE

// ---- FB/01_Axis/DUTs/ST_AxisState.TcDUT
TYPE ST_AxisState :
STRUCT
	uiNodeAddr									:UINT									;			//从站节点地址		
	rActModuloPos								:REAL									;			//实际位置-模轴位置
	rActPos										:REAL									;			//实际位置-线性位置
	rActVel										:REAL									;			//实际速度	
	rActAcc										:REAL									;			//实际加速度	
	rActTrq										:REAL									;			//实际扭矩	
	bDirPositive								:BOOL									;			//正向运动标志	
	bDirNegative								:BOOL									;			//负向运动标志	
	bPowerOK									:BOOL									;			//使能完成	
	bHoming										:BOOL									;			//回零中	
	bHome_OK									:BOOL									;			//回零完成	
	siModeOfOperation						    :SINT					                ;		    //  驱动器输出PLC工作模式，传递给PLC的工作模式	
	bPSw										:BOOL									;			//正极限	
	bNSw										:BOOL									;			//负极限	
	bHSw										:BOOL									;			//原点开关	
	bStandStill									:BOOL									;			//停止中
	bMoving										:BOOL									;			//移动中
	bHasJob                                     :BOOL									;			//工作中
	bInSync										:BOOL									;			//耦合中	
	bError										:BOOL									;			//报错
	bWarning									:BOOL									;			//警告
	bLightEror									:BOOL									;			//轻量错误
	bCriticalError								:BOOL									;			//严重错误
	arErrorID									:ARRAY[1..12] OF BOOL					;			//错误ID
	udiNCErrorID								:UDINT									;			//NC ErrorID
	uiDriveErrorCode							:UINT									;			//驱动器报警代码
END_STRUCT	
END_TYPE

// ---- FB/01_Axis/DUTs/ST_HomeViaDrivePar.TcDUT
TYPE ST_HomeViaDrivePar :
STRUCT
	//必须设定的参数
//	nCtrl1					AT%I*			:				USINT					;				// 驱动器回零模式下配置 : NC输出的控制字1，传递给PLC 
//	nCtrl2					AT%I*			:				USINT					;				// 驱动器回零模式下配置 : NC输出的控制字1，传递给PLC 
//	ControlWord				AT%Q*			:				UINT					;				// 驱动器回零模式下配置 : PLC输出控制字，传递给驱动器的控制字 
	ModeOfOperation			AT%Q*			:				SINT					;				// 驱动器回零模式下配置 : PLC输出驱动器工作模式，传递给驱动器的工作模式		
	//根据驱动器的实际需求进行设置
	siHomeMethod							:				SINT					;				// 设置通过驱动器回零的方式
	udiHomeVelHigh							:				UDINT					;				// 设置通过驱动器回零的高速回零速度
	udiHomeVelLow							:				UDINT					;				// 设置通过驱动器回零的低速回零速度
	udiHomeAcc								:				UDINT					;				// 设置通过驱动器回零的加减速度
	diHomeOffset							:				DINT					;				// 设置通过驱动器回零的回零偏置
	rHomeVelHigh							:				LREAL					;				// 设置通过探针回零的高速回零速度
	rHomeVelLow							    :				LREAL					;				// 设置通过探针回零的低速回零速度
	rHomeOffset							    :				LREAL					;				// 设置通过探针回零的回零偏置
END_STRUCT
END_TYPE

// ---- FB/11_AIO/DUTs/ST_AIO.TcDUT
TYPE ST_AIO :
STRUCT
	rAI1				:			REAL			;			// 底部负压表显示
	rAI2				:			REAL			;			// 针头气压表显示
	rAI3				:			REAL			;			// 
	rAI4				:			REAL			;			// 
	rAI5				:			REAL			;			// 底部负压比例阀反馈
	rAI6				:			REAL			;			// 针头负压比例阀反馈
	rAI7				:			REAL			;			// 针头正压比例阀反馈
	rAI8				:			REAL			;			//
	rAI9				:			REAL			;			//
	rAI10				:			REAL			;			//
	rAI11				:			REAL			;			//
	rAI12				:			REAL			;			//
	rAI13				:			REAL			;			//
	rAI14				:			REAL			;			//
	rAI15				:			REAL			;			//
	rAI16				:			REAL			;			//
	rAI17				:			REAL			;			//
	rAI18				:			REAL			;			//
	rAI19				:			REAL			;			//
	rAI20				:			REAL			;			//

	rAO1				:			REAL			;			// 底部负压比例阀设定
	rAO2				:			REAL			;			// 针头负压比例阀设定
	rAO3				:			REAL			;			// 针头正压比例阀设定
	rAO4				:			REAL			;			//
	rAO5				:			REAL			;			//
	rAO6				:			REAL			;			//
	rAO7				:			REAL			;			//
	rAO8				:			REAL			;			//
	rAO9				:			REAL			;			//
	rAO10				:			REAL			;			//
	rAO11				:			REAL			;			//
	rAO12				:			REAL			;			//
	rAO13				:			REAL			;			//
	rAO14				:			REAL			;			//
	rAO15				:			REAL			;			//
	rAO16				:			REAL			;			//
END_STRUCT
END_TYPE

// ---- FB/31_PDMSCtr/DUTs/ST_LightCtr.TcDUT
TYPE ST_LightCtr :
STRUCT
	iChannel1ValueSet		:				UINT						;			//通道1设定值
	iChannel2ValueSet		:				UINT						;			//通道2设定值
	iChannel3ValueSet		:				UINT						;			//通道3设定值
	iChannel4ValueSet		:				UINT						;			//通道4设定值
	iChannel1ActValue		:				UINT						;			//通道1当前值
	iChannel2ActValue		:				UINT						;			//通道2当前值
	iChannel3ActValue		:				UINT						;			//通道3当前值
	iChannel4ActValue		:				UINT						;			//通道4当前值
END_STRUCT
END_TYPE

// ---- FB/02_NCI/DUTs/ST_IJP.TcDUT
TYPE ST_IJP :
STRUCT
	in_stItpToPlc AT %I*: NCTOPLC_NCICHANNEL_REF;
	out_stItpToPlc AT %Q*:  PLCTONC_NCICHANNEL_REF;
	strNciName			    :STRING(255)			    ;           // NCI通道名
	bBuildGroupExe			:BOOL				        ;			// 将NC轴添加进NCI通道中 —— 触发
	bClearGroupExe			:BOOL				        ;			// 清除NCI通道中的轴，释放轴 —— 触发
	bLoadPGMExe			    :BOOL				        ;			// G代码装载
	bStartExe			    :BOOL				        ;			// 启动NC通道
	bStopExe			    :BOOL				        ;			// 停止NC通道
	bEstopExe			    :BOOL				        ;			// 紧急停止NCI
	bItpEStopEx             : BOOL ;                                 //  暂停G代码
	bItpStepOnAfterEStopEx  : BOOL                    ;               //  继续G代码
	bAfterEstopExe			:BOOL				        ;			// 紧急停止后恢复
	bResetExe			    :BOOL				        ;			// 错误复位
	bWriteRParExe			:BOOL				        ;				// 写R变量
	bReadRParExe			:BOOL				        ;				// 读R变量
	bLayerChanging			:BOOL				        ;				// 图层切换标志
	bLayerChanged			:BOOL				        ;	       // 图层切换指令
	bPrintDone			    :BOOL				        ;           // 轨迹执行完成
	bLoadPGMDone			:BOOL				        ;    // load路径文件完成
	bEx_TrigH			    :BOOL				        ;		    // 高压触发	输出到硬件
    bEx_Trig			        :BOOL				        ;		    // 阀触发	输出到硬件	
	bEx_TrigHfb			              :BOOL				        ;		    // 手动高压触发	输出到硬件反馈
    bEx_Trigfb			              :BOOL				        ;		    // 手动阀触发	输出到硬件反馈	
    EL5131_CamCtrlMax       :int                        ;// 最大位置比较数组量	
	arrWriteRPar			:ARRAY[0..19] OF LREAL		;
	arrReadRPar			    :ARRAY[0..19] OF LREAL		;
    bEx_TrigEl5131          :BOOL				        ;		    // 位置比较触发允许		
    bWriteZeroShiftExe      :BOOL;
	bEx_TrigBumpBack		:BOOL;								//开泵回抽模式
	lZeroShiftX             :LREAL                      ;           //X偏移值
	lZeroShiftY             :LREAL                      ;           //Y偏移值
	lZeroShiftZ             :LREAL                      ;           //Z偏移值


	

    rPosTolerance           :LREAL :=0.01                     ;           //位置比较允许误差
	tEndPosDelay            :TIME   :=T#1S                       ;           //终点比较延迟时间
//	bTrigSwitch             :BOOL                       ;           //位置比较高压是否开启(on=开)
//	bTrigPreSwitch          :BOOL                       ;          //比置比较例阀是否开启(on=开)
		
    bEl5131_TrigH:  BOOL;                                         //  (1-X1/Y1/Z1位置触发) (2-X1/Y2/Z1位置触发) (3-X2/Y1/Z2位置触发) (4-X2/Y2/Z2位置触发)
    bEl5131_Trig :  BOOL;
 
	strPRGName			    :STRING(255)			    ;           // 文件名
	lrOverrideSet			:LREAL				        ;			// 速度比例设定
	iJetOnDelay			    :INT:=1						;			// 喷墨开延时
	iJetOffDelay			:INT						;			// 喷墨关延时

//	udiErrOutToPlc                  AT%I*                     :UDINT;            // NCI故障码
//    lrPathVeloOutToPlc              AT%I*                     :LREAL ;           // NCI合成速度
	arErrorID									:ARRAY[1..7] OF BOOL;			//错误ID
	udiError									:UDINT			    ;// 错误编号
	bError										:BOOL													;			// 错误标志
    bErrorEStop                                  : BOOL ;                    ;            //  G代码暂停错误标志
	
END_STRUCT
END_TYPE

// ---- FB/41_PosCom/DUTs/ST_EL5131_CamCtrl.TcDUT
TYPE ST_EL5131_CamCtrl :
STRUCT
    // ------------------- 输入变量（控制指令） -------------------
	rPosStart1				 :	LREAL;// 比较起点位置x
	rPosStart2				 :	LREAL;// 比较起点位置y
	rPosStart3				 :	LREAL;// 比较起点位置z
	rPosEnd1                 :	LREAL;// 比较终点位置x
	rPosEnd2                 :	LREAL;// 比较终点位置y
	rPosEnd3                 :	LREAL;// 比较终点位置z
	bCamCtrlStartEn                 :	BOOL;// 比较点执行许可标志
	bCamCtrlEndEn                   :	BOOL;// 比较点执行许可标志
	udiAxisId1               :UDINT                      ;           // 参与位置比较轴ID
	udiAxisId2               :UDINT                      ;           // 参与位置比较轴ID
	udiAxisId3               :UDINT                      ;           // 参与位置比较轴ID
END_STRUCT
END_TYPE

// ---- FB/61_Alarm/DUTs/Enum_ErrorClass.TcDUT
TYPE Enum_ErrorClass :
(
    NoAlarm                		:=0,					//无警报
    Message      				:=1,					//信息
    Event           			:=2,					//事件
    Reserve3		            :=3,					//预留
    Reserve4                   	:=4,					//预留
    Reserve5                   	:=5,					//预留
    LightError          		:=6,					//轻微报警
    CriticalError               :=7						//重度报警
);
END_TYPE

// ---- FB/61_Alarm/DUTs/ST_Error.TcDUT
TYPE ST_Error :
STRUCT
    (*InPut*)
	iErrorID					:					INT						;			//报警ID号
    wstrErrorMessage			:					WSTRING					;			//报警信息
    dtErrorOccorTime			:                   DT						;			//报警发生时间
	bErrorExe					:					BOOL					;			//报警触发信号接入
	bFilterOn					:					BOOL					;			//输入信号滤波功能
	timeFilter					:                   TIME					;			//滤波时间设定
	bResetSignalUse				:					BOOL					;			//启用复位信号复位.true=复位信号为1时且触发信号为0时，复位报警状态;  false=仅触发信号为0时复位报警信号
	bResetExe					:					BOOL					;			//报警复位信号接入
	enumErrorClass				:					Enum_ErrorClass			;			//报警等级

	bAlarmAction1				:					BOOL					;			//报警后输出动作1
	bAlarmAction2				:					BOOL					;			//报警后输出动作2
	bAlarmAction3				:					BOOL					;			//报警后输出动作3
	bAlarmAction4				:					BOOL					;			//报警后输出动作4

   (*OutPut*)
	bErrorOccur					:					BOOL					;			//报警正在发生
	bEnabled					:                	BOOL					;			//当前报警已启用
END_STRUCT
END_TYPE;

// ---- FB/61_Alarm/DUTs/ST_HistoryError.TcDUT
TYPE ST_HistoryError :
STRUCT
  	wstrErrorMessage				:            	WSTRING					;	//报警信息
	iErrorID						:				INT						;	//报警ID号
   	dtErrorTime						:               DT						;	//报警发生时间
END_STRUCT
END_TYPE

// ---- FB/71_Gear/DOUTs/ST_Gear.TcDUT
TYPE ST_Gear :
STRUCT
	wstrName		           :WSTRING	;
    AxisRefMaster  				: Axis_Ref;
	AxisRefSlave   				: Axis_Ref;			        
	bGearIn                     :BOOL;         // 耦合变量
	bFlyGearIn                  :BOOL;         //  飞剪耦合变量
	bGearOut                    :BOOL;         // 耦合变量
	bStop_A                     :BOOL;        //  运动停止
	rRatioNumerator           :LREAL;         // 从轴速度
	uiRatioDenominator        :UINT;         // 主轴速度
	bInSyncing                :BOOL;         // 耦合中
	bFlyInSyncing                :BOOL;         // 耦合中
	bnoInSyncing                 :BOOL;         // 解耦
	rMasterSyncPosition      :LREAL;         // 主轴同步位置
	rSlaveSyncPosition       :LREAL;         // 从轴同步位置
	rSyncVelocity            :LREAL;         // 同步最大速度
	rSyncACC                 :LREAL;
	rSyncDEC                 :LREAL;
	rSyncJerk                :LREAL;
	bError	                 :BOOL;          //  错误状态
	arErrorID				 :ARRAY[1..3] OF BOOL;			//错误ID
END_STRUCT
END_TYPE

// ---- GVLs/Com_GVLS.TcGVL

VAR_GLOBAL
   (* 结构体申明*)
   stSystem          : ST_System:=(strDeviceName:='EHD');
   arstAxis            : ARRAY[1..10] OF ST_Axis;  
   stIJP             : ST_IJP     := (strNciName:='C:\NC\1.nc',lrOverrideSet := LREAL#100);   
   stAIO             : ST_AIO;   
   stLightCtr        : ST_LightCtr;
   arstCamCtrlIO       : ARRAY[1..100] OF ST_EL5131_CamCtrl; //1-X轴 2-Y轴
   bPlatformVacON    :BOOL       :=FALSE;(*真空吸附*)
   bPlatformVacOff   :BOOL       :=FALSE;
   arstHomeADS          :ARRAY[1..10] OF ST_HomeAdsGroup;
   arstHomeCoE          :ARRAY[1..10] OF ST_HomeCoEGroup;
   arstYV					: ARRAY[1..15] OF ST_YV; //所有气缸定义   
   arstVac				:ARRAY[1..15] OF ST_Vacuum; //所有真空定义
   stPump				:ST_Pump;
   arstGear           :ARRAY[1..2] OF ST_Gear;
END_VAR

// ---- GVLs/GVL_ALM.TcGVL
VAR_GLOBAL
	//当前正在发生的警报数量
	iActErrorNum					:             		INT																;
	//历史发生的警报数量
	iHistoryErrorNum				:           		INT																;
	//报警信息数组，根据iErrorIDMax设定上限值。根据需求扩展。
	arrstError						:					ARRAY [1..iErrorIDMax] OF ST_Error								;
	//当前正在发生的报警存储数组，预设30组数据
	arrstActError					:					ARRAY [1..30] OF ST_HistoryError								;
	//清除历史报警信息数组触发变量
	bClearHistoryError				:            		BOOL															;
	//获取的当前系统时间，配合报警信息输出
	tActSystemTime					: 					TIMESTRUCT														;
	// 报警信息中英文选择，默认为中文
	bLanguageSet					:					BOOL															;
END_VAR
VAR_GLOBAL PERSISTENT
	//历史报警存储数组，预设200组数组
	arrstHistoryError				:					ARRAY [1..200] OF ST_HistoryError								;			
END_VAR
VAR_GLOBAL CONSTANT
	// 报警数组最大值，根据实际需求更改
	iErrorIDMax: INT := 500;
END_VAR
VAR_GLOBAL
	bGetSystemTimeDone: BOOL;
END_VAR

// ---- GVLs/GVL_IO.TcGVL
VAR_GLOBAL
(*X*)
	X000001  AT%I*:  BOOL;   // 急停
	X000002  AT%I*:  BOOL;   // X- NO
	X000003  AT%I*:  BOOL;   // x+ NO
	X000004  AT%I*:  BOOL;   // Y- NO
	X000005  AT%I*:  BOOL;   // y+ NO
	X000006  AT%I*:  BOOL;   // 
	X000007  AT%I*:  BOOL;   // 
	X000008  AT%I*:  BOOL;   // Z1+NC 
	X000009  AT%I*:  BOOL;   // Z1-NC 
	X000010  AT%I*:  BOOL;   // Z2+NC 
	X000011  AT%I*:  BOOL;   // Z2-NC 
	X000012  AT%I*:  BOOL;   // 
	X000013  AT%I*:  BOOL;   // 
	X000014  AT%I*:  BOOL;   // 
	X000015  AT%I*:  BOOL;   // 
	X000016  AT%I*:  BOOL;   // 
	
	X001001  AT%I*:  BOOL;   // R1+ 
	X001002  AT%I*:  BOOL;   // R1-
	X001003  AT%I*:  BOOL;   // R2+
	X001004  AT%I*:  BOOL;   // R2-
	X001005  AT%I*:  BOOL;   // R3+
	X001006  AT%I*:  BOOL;   // R3-
	X001007  AT%I*:  BOOL;   // BUMP+
	X001008  AT%I*:  BOOL;   // bump-
	X001009  AT%I*:  BOOL;   // 
	X001010  AT%I*:  BOOL;   // 
	X001011  AT%I*:  BOOL;   // 
	X001012  AT%I*:  BOOL;   // 
	X001013  AT%I*:  BOOL;   // 
	X001014  AT%I*:  BOOL;   // 
	X001015  AT%I*:  BOOL;   // 
	X001016  AT%I*:  BOOL;   // 
	
(*Y*)	
	Y000001 AT%Q*:  BOOL;   // 针头正负压切换阀
	Y000002 AT%Q*:  BOOL;   // 
	Y000003 AT%Q*:  BOOL;   // 
	Y000004 AT%Q*:  BOOL;   // 气缸开
	Y000005 AT%Q*:  BOOL;   //	气缸关 
	Y000006 AT%Q*:  BOOL;   // 	真空破1
	Y000007 AT%Q*:  BOOL;   //  真空吸1
	Y000008 AT%Q*:  BOOL;   //  真空破2
	Y000009 AT%Q*:  BOOL;   //  真空吸2
	Y000010 AT%Q*:  BOOL;   //  真空吸3
	Y000011 AT%Q*:  BOOL;   //  真空破3
	Y000012 AT%Q*:  BOOL;   // 
	Y000013 AT%Q*:  BOOL;   // 
	Y000014 AT%Q*:  BOOL;   // 
	Y000015 AT%Q*:  BOOL;   // 
	Y000016 AT%Q*:  BOOL;   // 高压输出
END_VAR

// ---- GVLs/Programdata.TcGVL
VAR_GLOBAL
	(* *******PTP/NCI*********** *)
	arAXIS:ARRAY[1..10] OF AXIS_REF;
	
	tonSystemFirstRun:TON;
	posEdgeFirstRun:R_TRIG;
	//in_stItpToPlc AT %I*:NCTOPLC_NCICHANNEL_REF;
	//out_stItpToPlc AT %Q*:PLCTONC_NCICHANNEL_REF;
	
	(* ******AIO****** *)	
	AX_1 AT%I*: ARRAY[1..4]  OF INT;// 根据3064、3062、3061情况确定数组长度
	AX_2 AT%I*: ARRAY[1..4]  OF INT;
	AY_1 AT%Q*: ARRAY[1..4]  OF INT;// 根据4004、4002情况确定数组长度
	AY_2 AT%Q*: ARRAY[1..4]  OF INT;

	(**************************************************************************)
	// stXDescPitch: ST_CompensationDesc := (fPosMin:=0.0, fPosMax:=100.0, nTableElements:=11)---安捷伦激光干涉仪补偿表取反,单位mm;
   stXPitchTable: ARRAY[0..20] OF ST_CompensationElement :=[(fPos:=0.0, fCompensation:=0.0),
                                                           (fPos:=10.0, fCompensation:=0.0),
                                                           (fPos:=20.0, fCompensation:=0.0),
                                                           (fPos:=30.0, fCompensation:=0.0),
                                                           (fPos:=40.0, fCompensation:=0.0),
                                                           (fPos:=50.0, fCompensation:=0.0),
                                                           (fPos:=60.0, fCompensation:=0.0),
                                                           (fPos:=70.0, fCompensation:=0.0),
                                                           (fPos:=80.0, fCompensation:=0.0),
                                                           (fPos:=90.0, fCompensation:=0.0),
                                                           (fPos:=100.0, fCompensation:=0.0),
                                                           (fPos:=110.0, fCompensation:=0.0),
                                                           (fPos:=120.0, fCompensation:=0.0),
                                                           (fPos:=130.0, fCompensation:=0.0),
                                                           (fPos:=140.0, fCompensation:=0.0),
                                                           (fPos:=150.0, fCompensation:=0.0),
                                                           (fPos:=160.0, fCompensation:=0.0),
                                                           (fPos:=170.0, fCompensation:=0.0),
                                                           (fPos:=180.0, fCompensation:=0.0),
                                                           (fPos:=190.0, fCompensation:=0.0),
                                                           (fPos:=200.0, fCompensation:=0.0)];
   //stYDescPitch: ST_CompensationDesc := (fPosMin:=0.0, fPosMax:=100.0, nTableElements:=11)---安捷伦激光干涉仪补偿表取反,单位mm;
   stYPitchTable: ARRAY[0..15] OF ST_CompensationElement :=[(fPos:=0.0, fCompensation:=0),
                                                           (fPos:=10.0, fCompensation:=-0.0),
                                                           (fPos:=20.0, fCompensation:=-0.0),
                                                           (fPos:=30.0, fCompensation:=-0.0),
                                                           (fPos:=40.0, fCompensation:=-0.0),
                                                           (fPos:=50.0, fCompensation:=-0.0),
                                                           (fPos:=60.0, fCompensation:=-0.0),
                                                           (fPos:=70.0, fCompensation:=-0.0),
                                                           (fPos:=80.0, fCompensation:=-0.0),
                                                           (fPos:=90.0, fCompensation:=-0.0),
                                                           (fPos:=100.0, fCompensation:=-0.0),
                                                           (fPos:=110.0, fCompensation:=-0.0),
                                                           (fPos:=120.0, fCompensation:=-0.0),
                                                           (fPos:=130.0, fCompensation:=-0.0),
                                                           (fPos:=140.0, fCompensation:=-0.0),
                                                           (fPos:=150.0, fCompensation:=-0.0)];
	(**************************************************************************) 
    
    (**)  
    bXProhibitFwMvALM		:			BOOL:=TRUE			;		(*	X 正向运动禁止报警*)
	bXProhibitBwMvALM		:			BOOL:=TRUE			;		(*	X 负向运动禁止报警*)
	
    bYProhibitFwMvALM		:			BOOL:=TRUE			;		(*	Y 正向运动禁止报警*)
	bYProhibitBwMvALM		:			BOOL:=TRUE			;		(*	Y 负向运动禁止报警*)
	
	bRProhibitFwMvALM		:			BOOL:=TRUE			;		(*	R 正向运动禁止报警*)
	bRProhibitBwMvALM		:			BOOL:=TRUE			;		(*	R 负向运动禁止报警*)
	
	bZ1ProhibitFwMvALM		:			BOOL:=TRUE			;		(*	Z1 正向运动禁止报警*)
	bZ1ProhibitBwMvALM		:			BOOL:=TRUE			;		(*	Z1 负向运动禁止报警*)
	
	bZ2ProhibitFwMvALM		:			BOOL:=TRUE			;		(*	Z2 正向运动禁止报警*)
	bZ2ProhibitBwMvALM		:			BOOL:=TRUE			;		(*	Z2 负向运动禁止报警*)
	
    (*从站号*)
    uiSlaveNum: UINT;
END_VAR

// ---- POUs/1_Axis/AxisLink.TcPOU
PROGRAM AxisLink
VAR
	fbAxis    :ARRAY[1..10] OF FB_Axis;//根据轴数量定义数组
	bFirstRun :BOOL;                  //上电初始化轴参数
	i         :INT;                   //用于轴报错
	fbAxisPECorect:ARRAY[1..2] OF FB_Axis_PE_Correct;
END_VAR

(*****************************************************************
1.轴PROG程序进行默认参数初始化并进行块调用及转system报错ID

2.	bPowerOn		     	// 伺服使能，置1操作,无自复位
    bHome_A				    // 回零,置1操作,无自复位
	bJogCw_A		        // 连续运动正向,上升沿作用,无自复位
	bJogCcw_A			    // 连续运动负向,上升沿作用,无自复位		
	bRelMove_A              // 相对移动,,上升沿作用,无自复位	
	bAbsMove_A              // 绝对移动,上升沿作用,无自复位	
	bStop_A				    // 自动停止,上升沿作用,自复位			
	bHomeStop               // 回零停止,上升沿作用,自复位	
	bReset_A			    // 复位,上升沿作用,自复位
	
3.	nCtrl1                  // link NC参数 --驱动回零轴，NC和驱动controlword通过程序关联 }
	nCtrl2                  // link NC参数 --驱动回零轴，NC和驱动controlword通过程序关联 }--控制字回零用
	ControlWord             // link PDO -- 6040,控制字                                   }
	ModeOfOperation         // link PDO -- 6060,模式切换
	iTorque                 // 设定扭矩 -- 6071,设定扭矩 

4.  uiMaxTorque 			// 最大扭矩     6072   onlineCOE,单位%
 	udiMaxVel 			    // 最大扭矩     607F   onlineCOE,单位P
 	HomeMethod              // 回零方法     6098   onlineCOE
    HomeOffset              // 回零偏置     607C   onlineCOE,单位P
 	HomSwitchVelo           // 驱动寻Z速度  6099.2 onlineCOE,单位P
  
5.	ModeOfOperationdis      // Readcoe-- 6061,控制模式反馈
	ActTorque 			    // Readcoe--6077 读取驱动器实际力矩 
	ErrorCode               // Readcoe-- 603F读取驱动器错误码   
	StatusWord              // Readcoe-- 6041 回零程序中驱动器状态字
	
6.  探针回零不使用上述2-5项配置
*****************************************************************)
(* 参数初始化*)
posEdgeFirstRun(CLK:=NOT bFirstRun);
IF posEdgeFirstRun.Q AND bFirstRun  =FALSE THEN;
arstAxis[1].Parameter.bAbsEnc:=FALSE;
arstAxis[1].Parameter.uiHomeMode:=8;
arstAxis[1].Parameter.bHmDir:=TRUE;
arstAxis[1].Parameter.sthomeViaDrivePar.diHomeOffset:=0;
//arstAxis[1].Parameter.sthomeViaDrivePar.siHomeMethod:=34;
arstAxis[1].Parameter.sthomeViaDrivePar.udiHomeVelHigh:=10;
arstAxis[1].Parameter.sthomeViaDrivePar.udiHomeVelLow:=5;
arstAxis[1].Parameter.sthomeViaDrivePar.udiHomeAcc:=3000;
arstAxis[1].Control.bHome_Con:=TRUE;
arstAxis[1].Parameter.rHmVel:=20;
arstAxis[1].Parameter.rJogVel_A:=100;
arstAxis[1].Parameter.rJogAcc_A:=3000;
arstAxis[1].Parameter.rJogDec_A:=3000;
arstAxis[1].Parameter.rStopDec:=30000;
arstAxis[1].Parameter.rStopJerk:=arstAxis[1].Parameter.rStopDec*50;
arstAxis[1].Parameter.sthomeViaDrivePar.ModeOfOperation:=8;
arstAxis[1].Control.bJogCw_Con:=TRUE;
arstAxis[1].Control.bJogCcw_Con:=TRUE;
arstAxis[1].Pos.Ctrl.bGo_Con:=TRUE;
arstAxis[1].Parameter.rInPosValue:=0.01;  // 到位阈值
arstAxis[1].Parameter.sthomeViaDrivePar.rHomeOffset:=0.0;
arstAxis[1].Parameter.sthomeViaDrivePar.rHomeVelHigh:=10.0;
arstAxis[1].Parameter.sthomeViaDrivePar.rHomeVelLow:=5.0;

arstAxis[2].Parameter.bAbsEnc:=FALSE;
arstAxis[2].Parameter.uiHomeMode:=8;
arstAxis[2].Parameter.bHmDir:=TRUE;
arstAxis[2].Parameter.sthomeViaDrivePar.diHomeOffset:=0;
//arstAxis[2].Parameter.sthomeViaDrivePar.siHomeMethod:=34;
arstAxis[2].Parameter.sthomeViaDrivePar.udiHomeVelHigh:=10;
arstAxis[2].Parameter.sthomeViaDrivePar.udiHomeVelLow:=5;
arstAxis[2].Parameter.sthomeViaDrivePar.udiHomeAcc:=3000;
arstAxis[2].Control.bHome_Con:=TRUE;
arstAxis[2].Parameter.rHmVel:=20;
arstAxis[2].Parameter.rJogVel_A:=100;
arstAxis[2].Parameter.rJogAcc_A:=3000;
arstAxis[2].Parameter.rJogDec_A:=3000;
arstAxis[2].Parameter.rStopDec:=30000;
arstAxis[2].Parameter.rStopJerk:=arstAxis[2].Parameter.rStopDec*10;
arstAxis[2].Parameter.sthomeViaDrivePar.ModeOfOperation:=8;
arstAxis[2].Control.bJogCw_Con:=TRUE;
arstAxis[2].Control.bJogCcw_Con:=TRUE;
arstAxis[2].Pos.Ctrl.bGo_Con:=TRUE;
arstAxis[2].Parameter.rInPosValue:=0.01;  // 到位阈值
arstAxis[2].Parameter.sthomeViaDrivePar.rHomeOffset:=0.0;
arstAxis[2].Parameter.sthomeViaDrivePar.rHomeVelHigh:=10.0;
arstAxis[2].Parameter.sthomeViaDrivePar.rHomeVelLow:=5.0;

arstAxis[3].Parameter.bAbsEnc:=FALSE;
arstAxis[3].Parameter.uiHomeMode:=0;
arstAxis[3].Parameter.bHmDir:=TRUE;
arstAxis[3].Control.bHome_Con:=TRUE;
arstAxis[3].Parameter.rHmVel:=20;
arstAxis[3].Parameter.rJogVel_A:=30;
arstAxis[3].Parameter.rJogAcc_A:=300;
arstAxis[3].Parameter.rJogDec_A:=300;
arstAxis[3].Parameter.rStopDec:=20000;
arstAxis[3].Parameter.rStopJerk:=arstAxis[3].Parameter.rStopDec*20;
arstAxis[3].Parameter.sthomeViaDrivePar.ModeOfOperation:=8;
arstAxis[3].Control.bJogCw_Con:=TRUE;
arstAxis[3].Control.bJogCcw_Con:=TRUE;
arstAxis[3].Pos.Ctrl.bGo_Con:=TRUE;
arstAxis[3].Parameter.sthomeViaDrivePar.rHomeOffset:=0.0;
arstAxis[3].Parameter.sthomeViaDrivePar.rHomeVelHigh:=2.0;
arstAxis[3].Parameter.sthomeViaDrivePar.rHomeVelLow:=1.0;

arstAxis[4].Parameter.bAbsEnc:=FALSE;
arstAxis[4].Parameter.uiHomeMode:=0;
arstAxis[4].Parameter.bHmDir:=TRUE;
arstAxis[4].Control.bHome_Con:=TRUE;
arstAxis[4].Parameter.rHmVel:=20;
arstAxis[4].Parameter.rJogVel_A:=30;
arstAxis[4].Parameter.rJogAcc_A:=300;
arstAxis[4].Parameter.rJogDec_A:=300;
arstAxis[4].Parameter.rStopDec:=20000;
arstAxis[4].Parameter.rStopJerk:=arstAxis[3].Parameter.rStopDec*20;
arstAxis[4].Parameter.sthomeViaDrivePar.ModeOfOperation:=8;
arstAxis[4].Control.bJogCw_Con:=TRUE;
arstAxis[4].Control.bJogCcw_Con:=TRUE;
arstAxis[4].Pos.Ctrl.bGo_Con:=TRUE;
arstAxis[4].Parameter.sthomeViaDrivePar.rHomeOffset:=0.0;
arstAxis[4].Parameter.sthomeViaDrivePar.rHomeVelHigh:=2.0;
arstAxis[4].Parameter.sthomeViaDrivePar.rHomeVelLow:=1.0;

arstAxis[5].Parameter.bAbsEnc:=FALSE;
arstAxis[5].Parameter.uiHomeMode:=0;
arstAxis[5].Parameter.bHmDir:=TRUE;
arstAxis[5].Control.bHome_Con:=TRUE;
arstAxis[5].Parameter.rHmVel:=20;
arstAxis[5].Parameter.rJogVel_A:=30;
arstAxis[5].Parameter.rJogAcc_A:=300;
arstAxis[5].Parameter.rJogDec_A:=300;
arstAxis[5].Parameter.rStopDec:=20000;
arstAxis[5].Parameter.rStopJerk:=arstAxis[3].Parameter.rStopDec*20;
arstAxis[5].Parameter.sthomeViaDrivePar.ModeOfOperation:=8;
arstAxis[5].Control.bJogCw_Con:=TRUE;
arstAxis[5].Control.bJogCcw_Con:=TRUE;
arstAxis[5].Pos.Ctrl.bGo_Con:=TRUE;
arstAxis[5].Parameter.sthomeViaDrivePar.rHomeOffset:=0.0;
arstAxis[5].Parameter.sthomeViaDrivePar.rHomeVelHigh:=2.0;
arstAxis[5].Parameter.sthomeViaDrivePar.rHomeVelLow:=1.0;

arstAxis[6].Parameter.bAbsEnc:=TRUE;
arstAxis[6].Parameter.uiHomeMode:=0;
arstAxis[6].Parameter.bHmDir:=TRUE;
arstAxis[6].Control.bHome_Con:=TRUE;
arstAxis[6].Parameter.rHmVel:=20;
arstAxis[6].Parameter.rJogVel_A:=30;
arstAxis[6].Parameter.rJogAcc_A:=300;
arstAxis[6].Parameter.rJogDec_A:=300;
arstAxis[6].Parameter.rStopDec:=20000;
arstAxis[6].Parameter.rStopJerk:=arstAxis[3].Parameter.rStopDec*20;
arstAxis[6].Parameter.sthomeViaDrivePar.ModeOfOperation:=8;
arstAxis[6].Control.bJogCw_Con:=TRUE;
arstAxis[6].Control.bJogCcw_Con:=TRUE;
arstAxis[6].Pos.Ctrl.bGo_Con:=TRUE;
arstAxis[6].Parameter.sthomeViaDrivePar.rHomeOffset:=0.0;
arstAxis[6].Parameter.sthomeViaDrivePar.rHomeVelHigh:=2.0;
arstAxis[6].Parameter.sthomeViaDrivePar.rHomeVelLow:=1.0;

arstAxis[7].Parameter.bAbsEnc:=FALSE;
arstAxis[7].Parameter.uiHomeMode:=0;
arstAxis[7].Parameter.bHmDir:=TRUE;
arstAxis[7].Control.bHome_Con:=TRUE;
arstAxis[7].Parameter.rHmVel:=20;
arstAxis[7].Parameter.rJogVel_A:=30;
arstAxis[7].Parameter.rJogAcc_A:=300;
arstAxis[7].Parameter.rJogDec_A:=300;
arstAxis[7].Parameter.rStopDec:=20000;
arstAxis[7].Parameter.rStopJerk:=arstAxis[3].Parameter.rStopDec*20;
arstAxis[7].Parameter.sthomeViaDrivePar.ModeOfOperation:=8;
arstAxis[7].Control.bJogCw_Con:=TRUE;
arstAxis[7].Control.bJogCcw_Con:=TRUE;
arstAxis[7].Pos.Ctrl.bGo_Con:=TRUE;
arstAxis[7].Parameter.sthomeViaDrivePar.rHomeOffset:=0.0;
arstAxis[7].Parameter.sthomeViaDrivePar.rHomeVelHigh:=2.0;
arstAxis[7].Parameter.sthomeViaDrivePar.rHomeVelLow:=1.0;
arstAxis[7].Parameter.uiAxisChannelNum:=1;


arstAxis[8].Parameter.bAbsEnc:=FALSE;
arstAxis[8].Parameter.uiHomeMode:=0;
arstAxis[8].Parameter.bHmDir:=TRUE;
arstAxis[8].Control.bHome_Con:=TRUE;
arstAxis[8].Parameter.rHmVel:=20;
arstAxis[8].Parameter.rJogVel_A:=30;
arstAxis[8].Parameter.rJogAcc_A:=300;
arstAxis[8].Parameter.rJogDec_A:=300;
arstAxis[8].Parameter.rStopDec:=20000;
arstAxis[8].Parameter.rStopJerk:=arstAxis[3].Parameter.rStopDec*20;
arstAxis[8].Parameter.sthomeViaDrivePar.ModeOfOperation:=8;
arstAxis[8].Control.bJogCw_Con:=TRUE;
arstAxis[8].Control.bJogCcw_Con:=TRUE;
arstAxis[8].Pos.Ctrl.bGo_Con:=TRUE;
arstAxis[8].Parameter.sthomeViaDrivePar.rHomeOffset:=0.0;
arstAxis[8].Parameter.sthomeViaDrivePar.rHomeVelHigh:=2.0;
arstAxis[8].Parameter.sthomeViaDrivePar.rHomeVelLow:=1.0;
arstAxis[8].Parameter.uiAxisChannelNum:=2;

arstAxis[9].Parameter.bAbsEnc:=FALSE;                                        
arstAxis[9].Parameter.uiHomeMode:=0;                                         
arstAxis[9].Parameter.bHmDir:=TRUE;                                          
arstAxis[9].Control.bHome_Con:=TRUE;                                         
arstAxis[9].Parameter.rHmVel:=20;                                            
arstAxis[9].Parameter.rJogVel_A:=30;                                         
arstAxis[9].Parameter.rJogAcc_A:=300;                                        
arstAxis[9].Parameter.rJogDec_A:=300;                                        
arstAxis[9].Parameter.rStopDec:=20000;                                        
arstAxis[9].Parameter.rStopJerk:=arstAxis[3].Parameter.rStopDec*20;          
arstAxis[9].Parameter.sthomeViaDrivePar.ModeOfOperation:=8;                  
arstAxis[9].Control.bJogCw_Con:=TRUE;                                        
arstAxis[9].Control.bJogCcw_Con:=TRUE;                                       
arstAxis[9].Pos.Ctrl.bGo_Con:=TRUE;                                          
arstAxis[9].Parameter.sthomeViaDrivePar.rHomeOffset:=0.0;                    
arstAxis[9].Parameter.sthomeViaDrivePar.rHomeVelHigh:=2.0;                   
arstAxis[9].Parameter.sthomeViaDrivePar.rHomeVelLow:=1.0;                    
arstAxis[9].Parameter.uiAxisChannelNum:=3;

arstAxis[10].Parameter.bAbsEnc:=FALSE;                                       
arstAxis[10].Parameter.uiHomeMode:=0;                                        
arstAxis[10].Parameter.bHmDir:=TRUE;                                         
arstAxis[10].Control.bHome_Con:=TRUE;                                        
arstAxis[10].Parameter.rHmVel:=1;                                           
arstAxis[10].Parameter.rJogVel_A:=1;                                        
arstAxis[10].Parameter.rJogAcc_A:=10;                                       
arstAxis[10].Parameter.rJogDec_A:=10;                                       
arstAxis[10].Parameter.rStopDec:=100;                                       
arstAxis[10].Parameter.rStopJerk:=arstAxis[3].Parameter.rStopDec*20;         
arstAxis[10].Parameter.sthomeViaDrivePar.ModeOfOperation:=8;                 
arstAxis[10].Control.bJogCw_Con:=TRUE;                                       
arstAxis[10].Control.bJogCcw_Con:=TRUE;                                      
arstAxis[10].Pos.Ctrl.bGo_Con:=TRUE;                                         
arstAxis[10].Parameter.sthomeViaDrivePar.rHomeOffset:=0.0;                   
arstAxis[10].Parameter.sthomeViaDrivePar.rHomeVelHigh:=1.0;                  
arstAxis[10].Parameter.sthomeViaDrivePar.rHomeVelLow:=1.0;                   

// 轴parameter地址
arstHomeADS[1].nCalibrationVel:=16#4001;
arstHomeADS[1].nHomeInfo:=16#5001;
arstHomeADS[2].nCalibrationVel:=16#4002;
arstHomeADS[2].nHomeInfo:=16#5002;
arstHomeADS[3].nCalibrationVel:=16#4003;
arstHomeADS[3].nHomeInfo:=16#5003;
arstHomeADS[4].nCalibrationVel:=16#4004;
arstHomeADS[4].nHomeInfo:=16#5004;
arstHomeADS[5].nCalibrationVel:=16#4005;
arstHomeADS[5].nHomeInfo:=16#5005;
arstHomeADS[6].nCalibrationVel:=16#4006;
arstHomeADS[6].nHomeInfo:=16#5006;

arstHomeADS[7].nCalibrationVel:=16#4007;
arstHomeADS[7].nHomeInfo:=16#5007;

arstHomeADS[8].nCalibrationVel:=16#4008;
arstHomeADS[8].nHomeInfo:=16#5008;

arstHomeADS[9].nCalibrationVel:=16#4009;
arstHomeADS[9].nHomeInfo:=16#5009;

arstHomeADS[10].nCalibrationVel:=16#400A;
arstHomeADS[10].nHomeInfo:=16#500A;

bFirstRun             :=TRUE;
END_IF
(* 轴块调用*)
A_01_AX();
A_02_AY();
A_03_AR();
A_04_AZ1();
A_05_AZ2();
A_06_APin();
A_07_R1();
A_08_R2();
A_09_R3();
A_10_Bump();
(* 轴补偿调用*)
fbAxisPECorect[1](
	AxisRef:= arAXIS[1], 
	arstPitchTable:= stXPitchTable, 
	bEnable:= , 
	bAxisHomeOK:= arstAxis[1].State.bHome_OK, 
	bBacklashDir:= , 
	rBcaklash:= , 
	rDistance:= 0, 
	lrCurBacklash=> , 
	lrCOmpensation=> , 
	bBusy=> , 
	bError=> );
(* 轴补偿调用*)
fbAxisPECorect[2](
	AxisRef:= arAXIS[2], 
	arstPitchTable:= stYPitchTable, 
	bEnable:= , 
	bAxisHomeOK:= arstAxis[2].State.bHome_OK, 
	bBacklashDir:= , 
	rBcaklash:= , 
	rDistance:= 0, 
	lrCurBacklash=> , 
	lrCOmpensation=> , 
	bBusy=> , 
	bError=> );

ACTION A_01_AX:
//Axis-BasicParameterSettings
// 限位默认常闭，常开需要取反,白色常开/黑色常闭
// 轴基础参数设定
arstAxis[1].wstrName:=" 喷涂X轴" ;
arstAxis[1].strNetID:=stSystem.strNetID;//'192.168.1.50.2.1';//arAXIS[1].DriveAddress.NetID;
//arstAxis[1].uiSlaveAddr; 通过drive-infoData-AMSNETID-PORT关联;
arstAxis[1].State.bNSw:= NOT  X000002 ;// PM-l25倍福接黑线，pmac接黑线 
arstAxis[1].State.bPSw:= NOT  X000003 ;


// 力矩
//stAxis[1].Parameter.uiMaxTorque:=800;
// 功能块
fbAxis[1](AxisRef:=arAXIS[1] , stAxis:=arstAxis[1] ,stHomeADS:=arstHomeADS[1], stHomeCoe:=arstHomeCoE[1],stSystem:=stSystem );
END_ACTION

ACTION A_02_AY:
//Axis-BasicParameterSettings
//限位默认常闭，常开需要取反,白色常闭/黑色常开
arstAxis[2].wstrName:=" 喷涂Y轴" ;
arstAxis[2].strNetID:=stSystem.strNetID;///'192.168.1.50.2.1';
//stAxis[2].Parameter.uiSlaveAddr:=1012;通过drive-infoData-AMSNETID-PORT关联;
arstAxis[2].State.bNSw:=NOT X000004 ;// NC-White
arstAxis[2].State.bPSw:=NOT X000005 ;//
//false=etercat
// 功能块
fbAxis[2](AxisRef:=arAXIS[2] , stAxis:=arstAxis[2] , stSystem:=stSystem , stHomeCoe:=arstHomeCoE[1],stHomeADS:=arstHomeADS[2]);
END_ACTION

ACTION A_03_AR:
//Axis-BasicParameterSettings
//限位默认常闭，常开需要取反,白色常闭/黑色常开
arstAxis[3].wstrName:=" 喷涂R轴" ;
arstAxis[3].strNetID:=stSystem.strNetID;//'192.168.1.50.2.1';
//arstAxis[3].Parameter.uiSlaveAddr:=1014;通过drive-infoData-AMSNETID-PORT关联;
arstAxis[3].State.bNSw:= X000014 ;// NC-White
//stAxis[3].State.bHSW:= X000013;
arstAxis[3].State.bPSw:= X000013 ;//
//false=etercat
// 功能块
fbAxis[3](AxisRef:=arAXIS[3] , stAxis:=arstAxis[3] , stSystem:=stSystem  , stHomeCoe:=arstHomeCoE[1],stHomeADS:=arstHomeADS[3]);
END_ACTION

ACTION A_04_AZ1:
//Axis-BasicParameterSettings
//限位默认常闭，常开需要取反,白色常闭/黑色常开
arstAxis[4].wstrName:=" 喷涂Z1轴" ;
arstAxis[4].strNetID:=stSystem.strNetID;//'192.168.1.50.2.1';
//arstAxis[4].Parameter.uiSlaveAddr:=1015;通过drive-infoData-AMSNETID-PORT关联;
arstAxis[4].State.bNSw:= X000009 ;// NC-White
arstAxis[4].State.bPSw:= X000008 ;//
//false=etercat
// 功能块
fbAxis[4](AxisRef:=arAXIS[4] , stAxis:=arstAxis[4] , stSystem:=stSystem  , stHomeCoe:=arstHomeCoE[1],stHomeADS:=arstHomeADS[4]);
END_ACTION

ACTION A_05_AZ2:
//Axis-BasicParameterSettings
//限位默认常闭，常开需要取反,白色常闭/黑色常开
arstAxis[5].wstrName:=" 喷涂Z2轴" ;
arstAxis[5].strNetID:=stSystem.strNetID;//'192.168.1.50.2.1';
//arstAxis[5].Parameter.uiSlaveAddr:=1016;通过drive-infoData-AMSNETID-PORT关联;
arstAxis[5].State.bNSw:= X000011 ;// NC-White
arstAxis[5].State.bPSw:= X000010 ;//
//false=etercat
// 功能块
fbAxis[5](AxisRef:=arAXIS[5] , stAxis:=arstAxis[5] , stSystem:=stSystem , stHomeCoe:=arstHomeCoE[1],stHomeADS:=arstHomeADS[5]);
END_ACTION

ACTION A_06_APin:
//Axis-BasicParameterSettings
//限位默认常闭，常开需要取反,白色常闭/黑色常开
arstAxis[6].wstrName:=" 顶pin轴" ;
arstAxis[6].strNetID:=stSystem.strNetID;//'192.168.1.50.2.1';
//arstAxis[6].Parameter.uiSlaveAddr:=1017;
arstAxis[6].State.bNSw:= TRUE ;// NC-White
arstAxis[6].State.bPSw:= TRUE;//
//false=etercat
// 功能块
fbAxis[6](AxisRef:=arAXIS[6] , stAxis:=arstAxis[6] , stSystem:=stSystem  , stHomeCoe:=arstHomeCoE[1],stHomeADS:=arstHomeADS[6]);
END_ACTION

ACTION A_07_R1:
//Axis-BasicParameterSettings
//限位默认常闭，常开需要取反,白色常闭/黑色常开
arstAxis[7].wstrName:=" R1轴" ;
arstAxis[7].strNetID:=stSystem.strNetID;//'192.168.1.50.2.1';
//arstAxis[7].Parameter.uiSlaveAddr:=1017;
arstAxis[7].State.bNSw:=X001002 (*X001001 *);// NC-White
arstAxis[7].State.bPSw:=X001001 (* X001002;*);//
//false=etercat
// 功能块
fbAxis[7](AxisRef:=arAXIS[7] , stAxis:=arstAxis[7] , stSystem:=stSystem , stHomeCoe:=arstHomeCoE[1],stHomeADS:=arstHomeADS[7]);
END_ACTION

ACTION A_08_R2:
//Axis-BasicParameterSettings
//限位默认常闭，常开需要取反,白色常闭/黑色常开
arstAxis[8].wstrName:=" R2轴" ;
arstAxis[8].strNetID:=stSystem.strNetID;//'192.168.1.50.2.1';
//arstAxis[8].Parameter.uiSlaveAddr:=1017;
arstAxis[8].State.bNSw:= X001004(*X001003 *);// NC-White
arstAxis[8].State.bPSw:= X001003 (*X001004*);//
//false=etercat
// 功能块
fbAxis[8](AxisRef:=arAXIS[8] , stAxis:=arstAxis[8] , stSystem:=stSystem  , stHomeCoe:=arstHomeCoE[1],stHomeADS:=arstHomeADS[8]);
END_ACTION

ACTION A_09_R3:
//Axis-BasicParameterSettings
//限位默认常闭，常开需要取反,白色常闭/黑色常开
arstAxis[9].wstrName:=" R3轴" ;
arstAxis[9].strNetID:=stSystem.strNetID;//'192.168.1.50.2.1';
//arstAxis[9].Parameter.uiSlaveAddr:=1017;
arstAxis[9].State.bNSw:= X001006(*X001005*) ;// NC-White
arstAxis[9].State.bPSw:= X001005(*X001006*);//
//false=etercat
// 功能块
fbAxis[9](AxisRef:=arAXIS[9] , stAxis:=arstAxis[9] , stSystem:=stSystem , stHomeCoe:=arstHomeCoE[1],stHomeADS:=arstHomeADS[9]);
END_ACTION

ACTION A_10_Bump:
//Axis-BasicParameterSettings
//限位默认常闭，常开需要取反,白色常闭/黑色常开
arstAxis[10].wstrName:=" Bump" ;
arstAxis[10].strNetID:=stSystem.strNetID;//'192.168.1.50.2.1';
//arstAxis[6].Parameter.uiSlaveAddr:=1017;
arstAxis[10].State.bNSw:= X001007 ;// NC-White
arstAxis[10].State.bPSw:= X001008;//
//false=etercat
// 功能块
fbAxis[10](AxisRef:=arAXIS[10] , stAxis:=arstAxis[10] , stSystem:=stSystem  , stHomeCoe:=arstHomeCoE[1],stHomeADS:=arstHomeADS[10]);
END_ACTION

END_PROGRAM

// ---- FB/01_Axis/FB/FB_Axis.TcPOU
FUNCTION_BLOCK FB_Axis
VAR_IN_OUT
	stAxis: ST_Axis;
	stSystem: ST_System;
	AxisRef: Axis_REF;
	stHomeADS:ST_HomeAdsGroup;
	stHomeCoe:ST_HomeCoEGroup;
END_VAR
VAR_INPUT

END_VAR
VAR
	strVersion: STRING;
	fbMcWritePosMonitorDisable: MC_WriteParameter;
	fbMcWritePosMonitorEnable: MC_WriteParameter;
	fbMcReadDistPerPulse: MC_ReadParameter;
	fbMcReadGearRatio: MC_ReadParameter;
	// 每脉冲移动量
	lrDistPerPulse: LREAL := 0.0001;
	// 减速比
	lrGearRatio: LREAL := 1;
	bySubIndex: BYTE;
	wIndex: WORD;
	bReadActPos0x6064: BOOL;
	fbEcCoESdoReadActPos: FB_EcCoESdoRead;
	blink100ms: BLINK;
	fbEcCoeSdoReadExDriveOp: FB_EcCoeSdoReadEx;
	strAxisName: STRING;
	bMoveBaseCon: BOOL;
	fbMcSetPos: MC_SetPosition;
	bHomeExe: BOOL;
	bReset: BOOL;
	bHoming: BOOL;
	bPowerOk:BOOL;
	// 1-定位运动
	// 2-JOG
	// 3-回零
	// 4-轴置位
	// 5-轴停止
	uiMotionCMD: UINT;
	fbDriveErrorCode: FB_EcCoESdoRead;
	tonPowerOn: TON;
	RtrigPowerOn: R_TRIG;
	mcPower: MC_Power;
	mcReadStatus: MC_ReadStatus;
	mcReset: MC_Reset;
	mcHMJog: MC_Jog;
	mcHMJogInching: MC_Jog;
	rHMJogVel: REAL;
	mcJogContinuous: MC_Jog;
	mcJogInching: MC_Jog;
	mcHomeP: MC_Home;
	mcHomeN: MC_Home;
	mcHmAbsMove: MC_MoveAbsolute;
	bHomed: BOOL;
	bHomeStop: BOOL;
	bHomeCMD: BOOL;
	bHomeCMDLast: BOOL;
	iHomeStep: INT;
	bHomeJogFExe: BOOL;
	bHomeJogBExe: BOOL;
	lrHomeOffset: LREAL;
	bJogFExe: BOOL;
	bJogBExe: BOOL;
	bPosUpdate: BOOL;
	bRelMoveCon: BOOL;
	bAbsMoveCon: BOOL;
	bPosCmd: BOOL;
	bMoveAbsExe: BOOL;
	bMoveRelExe: BOOL;
	iPosId: INT;
	// 相对运动初始位置
	rRelStartPos: REAL;
	rVelEx: REAL;
	rPosEx: REAL;
	bRelEx: BOOL;
	rAccEx: REAL;
	rDecEx: REAL;
	rJerkEx: REAL;
	rVelExTmp: REAL;
	eDirection: MC_DIRECTION;
	iPosInstNum: INT;
	bPosDone1: BOOL;
	bPosDone2: BOOL;
	bPosBusy1: BOOL;
	bPosBusy2: BOOL;
	fbMC_MoveA: MC_MoveAbsolute;
	fbMC_MoveA2: MC_MoveAbsolute;
	fbMC_MoveR: MC_MoveRelative;
	fbMC_MoveR2: MC_MoveRelative;
	TonAxisMove: TON;
	lrStopMoveDec: LREAL;
	bStopMoveExe: BOOL;
	bStopExe: BOOL;
	fbMcStop: MC_Stop;
	bResetLast: BOOL;
	bWrongDirection: BOOL;
	bTouchProbeEnable: BOOL;
	w60B9: WORD;
	RtrigTouchDone: R_TRIG;
	Ton01: TON;
	diTouchCatchPos: DINT;
	bHomeSetPos: BOOL;
	MC_SetPosHome: MC_SetPosition;
	Ton06: TON;
	Ton05: TON;
	Ton03: TON;
	Ton04: TON;
	Ton02: TON;
	bMoveZeroPos: BOOL;
	MC_MoveZeroHome: MC_MoveAbsolute;
	bStopMoveExeLast: BOOL;
	m: INT;
	RtrigJogF: R_TRIG;
	RtrigJogB: R_TRIG;
	bHomeJogInchingFExe: BOOL;
	TonWaitStandStill: TON;
	blink10ms: BLINK;
	bSDOExe: BOOL := true;
	Ton07: TON;
	uiStatusWord: UINT;
	FB_EcCoESdoRead_6041: FB_EcCoESdoRead;
	// 修改驱动器工作字
	FB_EcCoESdoWrite_6060: FB_EcCoESdoWrite;
	siOldModeOfOperation: SINT;
	// 定位运动完成中间变量
	bGo_OK: BOOL;
	TonReadDriveErrorCode: TON;
	arrfbSetAlarm: ARRAY[1..12] OF FB_SetError;
	FB_EcCoESdoWrite_6098: FB_EcCoESdoWrite;
	FB_EcCoESdoWrite_6099_01: FB_EcCoESdoWrite;
	FB_EcCoESdoWrite_6099_02: FB_EcCoESdoWrite;
	FB_EcCoESdoWrite_609A: FB_EcCoESdoWrite;
	FB_EcCoESdoWrite_607C: FB_EcCoESdoWrite;
	siOldHomeMethod: SINT;
	udiOldHomeVelHigh: UDINT;
	udiOldHomeVelLow: UDINT;
	udiOldHomeAcc: UDINT;
	udiHomeVelHigh: UDINT;
	udiHomeVelLow: UDINT;
	udiHomeAcc: UDINT;
	Ton61: TON;
	bPosMonitorDisabled: BOOL;
	bPosMonitorAbled: BOOL;
	bSDO: BOOL;
	Ton62: TON;
	strDriveAddressNetID: STRING;
	uiDriveAddressSlaveAddr: UINT;
	mcReadDriveAddress: MC_ReadDriveAddress;
	tonReadDriveAddr: TON;
	bInitDone: BOOL;
	diHomeOffset: DINT;
	fbEcCoeSdoWriteExTargetTrq: FB_EcCoeSdoWriteEx;
	iTorqueTemp: INT;
	iTorqueTempOld: INT;
	iHomeStepPre: INT;
	FBTouchProbeHomeBylimit:FB_TouchProbe_Home_Bylimit;
	FBDriveHome:FB_Drive_Home;
	
END_VAR

 (*********
 	by Yu
	
	2023-12-15  1-增加 带绝对值编码器运动轴的回零标志位，默认一直存在原点。
				2-根据模轴或线性轴，输出当前位置。
	2023-12-19  增加置位功能	
	2023-12-26 	1-增加参数读取功能，分别读取当前轴设定的分辨率和减速比参数，探针回零时使用
				2-增加轴运行模式读取设定功能，通过COE实现。默认CSP模式。
				3-将wIndex、bySubIndex变量由外部轴变量转换为内部变量			
	2024-1-2	1-增加是否EtherCAT总线控制轴的判断，EtherCAT总线控制轴方可通过COE更换运行模式。	
				2-EtherCAT总线轴运行模式切换，松下电机需要取消 0x6060 的映射。
							
	2024-2-21	增加回零模式-4旋转寻Z相回零中，回零开始前移出Z相位置，同时增加寻Z相完成后等待到位时间
	2024-3-29	轴参数结构体中增加模轴当前位置变量 rActModuloPos ，同时分别输出模轴位置和线性位置
	2024-4-11	更改轴报警信息
	2024-4-15	增加回零模式5------碰硬限位回零，根据转矩判断
	2024-4-16	增加 MC_ReadDriveAddress 读取轴ADS参数，无需外部写入设定。
	2024-4-28	增加NC ErrorID输出，驱动器报警错误码输出,取消输出变量udiErrorID
	2024-5-7	优化碰硬限位回零模式，重新上使能，处理力矩问题
	2024-5-31	增加版本更新时间记录变量
	2024-06-04	将JOG运行，HOME运行，Pos运行的运行条件Con写入首次运行中，不在外部额外写入，外部根据实际需求写。
	2024-06-22	增加回零模式6 ---- 驱动器回零模式
	2024-06-24	屏蔽未上使能报警
	2024-07-05  增加回零模式6下，非回零状态，将运行模式写成8-CSP模式。
	2024-07-27	定位运动，绝对式运行，增加到位信号 的判定条件 - 位置比对：当前值与设定值偏差不超过 0.01 
	2024-08-15	到位判断，位置偏差参数开放。初始值为 0.01
	2024-08-16	增加定位完成中间变量 ，与位置偏差判断共同输出到位完成信号
				取消可变数组，只允许走9个位置
	2024-08-17	停止信号进入，清楚 定位运动中的 moving 信号，以及 iposId
				驱动器报警增加延时，先读取报警code，50ms后输出
	2024-08-20	增加回零流程开始时，复位回零功能块
	2025-02-06	增加复位触发信号
				功能块整理为多个Action。
	2025-03-14	增加程序可读性,取消9个位置存储方式。只支持走一个位置。后续可通过不断刷入位置来实现走多个位置。
				增加相对运动位置到位判断
				修改多次定位，在相对位置运动下不支持多次定位,只有在绝对位置运动下支持多次定位。
	2025-03-26	取消对力矩模式切换的控制
	2025-03-27	针对多轴驱动器，增加映射偏置
	2025-07-23	改写轴报警输出功能，轴报警预设存储于数组 101 起，每轴预留 12 个报警位
				修改当前功能块轴报警 ID 从 1 到 12，共计 12 组报警数据（空余一组）。
	2025-08-04	修改回零模式 6 -通过驱动器回零。整合驱动器回零需要的参数。
					1.删去 StatusWord , nState1 , nState2变量。删去 iPDO_6071（目标转矩）变量（后续需要可直接SDO读写）
					2.打包驱动器回零需设置的参数变量，集合到一个结构体中：
						a. 需要映射的变量 nCtrl1 , nCtrl2 , ControlWord . 控制值，分别映射 实际轴和 NC轴。
						b. ModeOfOperatiion变量，尽量通过映射修改。如果驱动器的 PDO 不支持修改，采用SDO读写方式。
						c. 新增参数 ———— 回零模式，回零速度（高、低速），回零加速度参数的设置。
				删去回零模式 5 - 碰硬档根据力矩回零。在驱动器中直接设置这种回零模式，倍福设置回零模式 6 。
	2025-08-05	更改 Init ，获取轴信息完成后，结束初始化。
	2025-08-08 	新增驱动器回零模式下，对 home offset 参数的设置
	2025-08-29	更新报警序号
	2025-09-04	修改单原点回零。回零启动步序设置为5。停止按钮按下，同步清除 bJogHomeBExe/bJogHomeFExe 的信号。
	2025-09-05	修改报警代码的映射范围。ErrorID 101 开始
	2025/09/10	增加定位运动的判断。绝对定位时，目标位置和当前位置之差小于判定窗口，不移动，直接输出到位信号
	2025/10/30	取消回零模式 3、4，需要进行Z相回零时，选用回零模式6-驱动器回零处理。
	2026/04/10	增加驱动器工作模式读取，存入对应变量 stAxis.State.siDriveOperationMode
				增加力矩设定程序。上位机写入参数值到 rTorque 中，程序中转换后写入 6071
	2026/04/15	回零模式6-驱动器回零，回零完成后，增加读取6064，并将6064的值换算后写入NC位置中操作。
	2025/04/21  回零模式6-驱动器回零。
				针对限位未接入驱动器内的回零模式，增加变量，可控制轴在驱动器回零前先移动到对应的限位处,再根据需求搜寻Z相。
				stAxis.Parameter.bHmDir 变量用于同步驱动器回零搜寻方向。
				stAxis.Parameter.sthomeViaDrivePar.bMoveToLimit 变量用于设定是否执行先移动到限位的操作。
				stAxis.Parameter.rHmVel 变量用于设置移动到限位的速度.
				
***********)
//当前版本更新时间
strVersion := '2026/04/21' ;


//
IF NOT bInitDone THEN
	A_01_Init();
ELSE
	A_02_StateIn();
	A_03_PowerOn();
	A_04_Reset();
	A_05_SetPos();
	A_06_Home();
	A_07_Jog();
	A_08_Move();
	A_09_Stop();
	A_11_StateOut();
	A_10_TrqCtr();
	A_12_Error();
END_IF;

ACTION A_01_Init:
{region "初始化"}
//模块首次运行，数据初始化 
bHomeCmd:=FALSE;
bHomeCmdLast:=FALSE;
	 
stAxis.Control.bHome_Con:=TRUE;
stAxis.Control.bJogCcw_Con:=TRUE;
stAxis.Control.bJogCw_Con:=TRUE;

//速度不允许非正数		 
IF stAxis.Parameter.rHmVel <= 0 THEN
	stAxis.Parameter.rHmVel:= 5;
END_IF;
IF stAxis.Parameter.rHmAcc <= 0 THEN
	stAxis.Parameter.rHmAcc:= 50;
END_IF;
IF stAxis.Parameter.rHmDec <= 0 THEN
	stAxis.Parameter.rHmDec:= 50;
END_IF;
IF stAxis.Parameter.rHmJerk <= 0 THEN
	stAxis.Parameter.rHmJerk:= 500;
END_IF;	
IF stAxis.Parameter.rJogVel_M <= 0 THEN
	stAxis.Parameter.rJogVel_M := 10;
END_IF;
IF stAxis.Parameter.rJogVel_A <= 0 THEN
	stAxis.Parameter.rJogVel_A := 10;
END_IF;	
IF stAxis.Parameter.rJogAcc_M <= 0 THEN
	stAxis.Parameter.rJogAcc_M := 100;
END_IF;	
IF stAxis.Parameter.rJogAcc_A <= 0 THEN
	stAxis.Parameter.rJogAcc_A := 100;
END_IF;	
IF stAxis.Parameter.rJogDec_M <= 0 THEN
	stAxis.Parameter.rJogDec_M := 100;
END_IF;	
IF stAxis.Parameter.rJogDec_A <= 0 THEN
	stAxis.Parameter.rJogDec_A := 100;
END_IF;	

stAxis.Parameter.rStopDec := 100000;
 
stAxis.Parameter.sthomeViaDrivePar.ModeOfOperation:=8;

		 
	stAxis.Parameter.rInPosValue := REAL#0.01 ;	
	  
	stAxis.Pos.Ctrl.bGo_Con:=TRUE;
	stAxis.Pos.Par.rVel:= 10;
	stAxis.Pos.Par.rAcc:= 100;
	stAxis.Pos.par.rDec:=100;
	stAxis.Pos.Par.rJerk:=1000;

	tonReadDriveAddr(IN:=TRUE , PT:=TIME#100MS , Q=> , ET=> );	 
	mcReadDriveAddress(
	Axis:= AxisRef, 
	Execute:= tonReadDriveAddr.Q  , 
	Done=> bInitDone , 
	Busy=> , 
	Error=> , 
	ErrorID=> , 
	DriveAddress=> );	 

{endregion}
END_ACTION

ACTION A_02_StateIn:
{region "状态读取”}
fbMcReadDistPerPulse(
	Axis:=AxisRef , 
	Enable:=tonPowerOn.Q , 
	ParameterNumber:=AxisEncoderScalingNumerator , 
	ReadMode:=READMODE_ONCE , 
	Value=>lrDistPerPulse );

fbMcReadGearRatio(
	Axis:= AxisRef, 
	Enable:=tonPowerOn.Q , 
	ParameterNumber:= AxisEncoderScalingDenominator,
	ReadMode:=READMODE_ONCE , 
	Value=>lrGearRatio );
	 
mcReadStatus(
	Axis:= AxisRef, 
	Enable:= TRUE, 
	Valid=> , 
	Busy=> , 
	Error=> , 
	ErrorID=> , 
	ErrorStop=> , 
	Disabled=> , 
	Stopping=> , 
	StandStill=> , 
	DiscreteMotion=> , 
	ContinuousMotion=> , 
	SynchronizedMotion=> , 
	Homing=> , 
	ConstantVelocity=> , 
	Accelerating=> , 
	Decelerating=> , 
	Status=> );

stAxis.Parameter.rInPosValue := ABS(stAxis.Parameter.rInPosValue);	 
	 
//延时读取
blink100ms(ENABLE:=TRUE,TIMELOW:=TIME#100MS,TIMEHIGH:=TIME#100MS);

//轴状态读取
stAxis.State.bStandStill := (AxisRef.Status.StandStill OR AxisRef.Status.NotMoving);
stAxis.State.bInSync := AxisRef.Status.SynchronizedMotion;
stAxis.State.bMoving := AxisRef.Status.Moving OR (stAxis.Parameter.uiHomeMode = 6 AND stAxis.State.bHoming) ;
stAxis.State.bDirPositive := AxisRef.Status.PositiveDirection;
stAxis.State.bDirNegative := AxisRef.Status.NegativeDirection;
stAxis.State.udiNCErrorID := AxisRef.Status.ErrorID;	 
	 
strDriveAddressNetID 	:=stAxis.strNetID;// AxisRef.DriveAddress.NetID ;
uiDriveAddressSlaveAddr :=stAxis.uiSlaveAddr;// AxisRef.DriveAddress.SlaveAddress ;

fbDriveErrorCode(
	sNetId:=strDriveAddressNetID  , 
	nSlaveAddr:=uiDriveAddressSlaveAddr , 
	nSubIndex:=16#00 , 
	nIndex:=(16#603F + (stAxis.Parameter.uiAxisChannelNum - 1)*16#800), 
	pDstBuf:= ADR(stAxis.State.uiDriveErrorCode) , 
	cbBufLen:=SIZEOF(stAxis.State.uiDriveErrorCode) , 
	bExecute:= AxisRef.Status.DriveDeviceError , 
	tTimeout:= , 
	bBusy=> , 
	bError=> , 
	nErrId=> , 
	cbRead=> );
		 
wIndex:=16#6064 + (stAxis.Parameter.uiAxisChannelNum - 1)*16#800;		  
bySubIndex:=16#00;

fbEcCoeSdoReadExDriveOp(
	sNetId:= strDriveAddressNetID , 
	nSlaveAddr:= uiDriveAddressSlaveAddr, 
	nSubIndex:= 16#00 , 
	nIndex:= (16#6061 + (stAxis.Parameter.uiAxisChannelNum - 1)*16#800), 
	pDstBuf:= ADR(stAxis.State.siModeOfOperation), 
	cbBufLen:= SIZEOF(stAxis.State.siModeOfOperation), 
	bExecute:= blink100ms.OUT, 
	tTimeout:= , 
	bCompleteAccess:= , 
	bBusy=> , 
	bError=> , 
	nErrId=> , 
	cbRead=> );

FB_EcCoESdoWrite_6060(
	sNetId:= strDriveAddressNetID, 
	nSlaveAddr:=uiDriveAddressSlaveAddr  , 
	nSubIndex:=16#00 , 
	nIndex:=16#6060 + (stAxis.Parameter.uiAxisChannelNum - 1)*16#800 , 
	pSrcBuf:=ADR(stAxis.Parameter.sthomeViaDrivePar.ModeOfOperation) , 
	cbBufLen:=SIZEOF(stAxis.Parameter.sthomeViaDrivePar.ModeOfOperation) , 
	bExecute:=siOldModeOfOperation <> stAxis.Parameter.sthomeViaDrivePar.ModeOfOperation , 
	tTimeout:= , 
	bBusy=> , 
	bError=> , 
	nErrId=> );
		 
siOldModeOfOperation := stAxis.Parameter.sthomeViaDrivePar.ModeOfOperation ;	 	
{endregion}
END_ACTION

ACTION A_03_PowerOn:
{region "使能&功能切换"}	 
	 		  
//运动条件
bMoveBaseCon := stAxis.State.bPowerOK AND NOT stAxis.State.bHoming AND NOT stAxis.State.bError AND NOT  stSystem.bEMG;
	
//运动功能切换（位置模式）
IF stAxis.State.bStandStill  THEN 
	IF stAxis.Pos.Ctrl.bGo_A OR (stAxis.Pos.Ctrl.bGo_M AND stSystem.bManual) THEN
		uiMotionCMD:=1;	
	ELSIF stAxis.Control.bJogCw_A OR (stAxis.Control.bJogCw_M AND stSystem.bManual) THEN
		uiMotionCMD := 2;
	ELSIF stAxis.Control.bJogCcw_A OR (stAxis.Control.bJogCcw_M AND stSystem.bManual) THEN
		uiMotionCMD :=2;
	ELSIF (stAxis.Control.bHome_A OR (stAxis.Control.bHome_M AND stSystem.bManual)) AND NOT stAxis.Parameter.bAbsEnc THEN
		uiMotionCMD :=3;
	ELSIF stAxis.Control.bSetPos THEN
		uiMotionCMD := 4;
	END_IF;		
END_IF;

	 
		  
//伺服使能
	tonPowerOn(
	IN:=stAxis.Control.bPowerOn AND NOT AxisRef.Status.DriveDeviceError AND NOT stSystem.bEMG  ,
	PT:=TIME#1MS);
	
    mcPower(
	Axis:= AxisRef, 
	Enable:=tonPowerOn.Q , 
	Enable_Positive:= stAxis.State.bPSW OR stAxis.State.bHoming , (* 撞限位高电平*)
	Enable_Negative:= stAxis.State.bNSW OR stAxis.State.bHoming, (* 撞限位高电平*)
	Override:= 100, 
	BufferMode:= , 
	Options:= , 
	Status=> stAxis.State.bPowerOK, 
	Busy=> , 
	Active=> , 
	Error=> , 
	ErrorID=> );

//mcPower(
//	Axis:= AxisRef, 
//	Enable:=tonPowerOn.Q , 
//	Enable_Positive:= TRUE , 
//	Enable_Negative:= TRUE , 
//	Override:= , 
//	BufferMode:= , 
//	Options:= , 
//	Status=>stAxis.State.bPowerOK , 
//	Busy=> , 
//	Active=> , 
//	Error=> , 
//	ErrorID=> );				
{endregion}
END_ACTION

ACTION A_04_Reset:
{region "轴复位"}	
mcReset(
	Axis:= AxisRef, 
	Execute:= (stSystem.bReset  OR stAxis.Control.bReset_A OR (stAxis.Control.bReset_M AND stSystem.bManual)) , 
	Done=> , 
	Busy=> , 
	Error=> , 
	ErrorID=> );
IF mcReset.Done OR mcReset.Error THEN
	stSystem.bReset:=FALSE;
	stAxis.Control.bReset_A:=FALSE;	 
   stAxis.Control.bReset_M:=FALSE;
END_IF;	
{endregion}
END_ACTION

ACTION A_05_SetPos:
{region"轴置位"}
IF uiMotionCMD = 4 THEN
	fbMcSetPos(
		Axis:=AxisRef , 
		Execute:= stAxis.Control.bSetPos AND bMoveBaseCon , 
		Position:= stAxis.Parameter.rSetPos, 
		Mode:= , 
		Options:= , 
		Done=> , 
		Busy=> , 
		Error=> , 
		ErrorID=> );
	
	stAxis.Control.bSetPos := FALSE;
END_IF 
{endregion}
END_ACTION

ACTION A_06_Home:
{region  "轴回零"}
//回零	
IF  (uiMotionCMD = 3) AND (NOT stAxis.Parameter.bAbsEnc) THEN
CASE stAxis.Parameter.uiHomeMode OF
	0:// 限位回零
	  FBTouchProbeHomeBylimit.bCMD_StartHomeIndex:=FALSE;
      IF stAxis.Parameter.bHmDir=TRUE THEN
		FBTouchProbeHomeBylimit.eCMD_HomeDirection:=MC_Negative_Direction;
	  ELSE
		FBTouchProbeHomeBylimit.eCMD_HomeDirection:=MC_Positive_Direction;	   
	  END_IF
	  FBTouchProbeHomeBylimit(
	    bCMD_HomeExecute:= stAxis.Control.bHome_A, 
	    bCMD_Reset:= stAxis.Control.bReset_A, 
	    bCMD_EnableState:= stAxis.State.bPowerOK, 
	    bCMD_StartHomeIndex:= , 
	    eCMD_HomeDirection:= , 
	    bCMD_PositiveLimit:= NOT stAxis.State.bPSw , 
	    bCMD_NegativeLimit:= NOT stAxis.State.bNSw, 
	    rCMD_HomePosition:= stAxis.Parameter.sthomeViaDrivePar.rHomeOffset, 
	    rCMD_TowardsVelSetValue:= stAxis.Parameter.sthomeViaDrivePar.rHomeVelHigh, 
	    rCMD_OffVelSetValue:= stAxis.Parameter.sthomeViaDrivePar.rHomeVelLow, 
	    stHomeAdsGroup:= stHomeADS, 
	    bResult_HomeDone=> stAxis.State.bHome_OK, 
	    bResult_HomeBusy=> stAxis.State.bHoming, 
	    bResult_HomeError=>(*stAxis.State.arErrorID[10]*), 
	    nResult_HomeErrorID=> , 
	    axis:=AxisRef );
    6:// 驱动回零
	
    8:// 倍福探针回零
      FBTouchProbeHomeBylimit.bCMD_StartHomeIndex:=TRUE;
      IF stAxis.Parameter.bHmDir=TRUE THEN
		FBTouchProbeHomeBylimit.eCMD_HomeDirection:=MC_Negative_Direction;
	  ELSE
		FBTouchProbeHomeBylimit.eCMD_HomeDirection:=MC_Positive_Direction;	   
	  END_IF
	  FBTouchProbeHomeBylimit(
	    bCMD_HomeExecute:= stAxis.Control.bHome_A , 
	    bCMD_Reset:= stAxis.Control.bReset_A, 
	    bCMD_EnableState:= stAxis.State.bPowerOK, 
	    bCMD_StartHomeIndex:= , 
	    eCMD_HomeDirection:= , 
	    bCMD_PositiveLimit:= NOT stAxis.State.bPSw , 
	    bCMD_NegativeLimit:= NOT stAxis.State.bNSw, 
	    rCMD_HomePosition:= stAxis.Parameter.sthomeViaDrivePar.rHomeOffset, 
	    rCMD_TowardsVelSetValue:= stAxis.Parameter.sthomeViaDrivePar.rHomeVelHigh, 
	    rCMD_OffVelSetValue:= stAxis.Parameter.sthomeViaDrivePar.rHomeVelLow, 
	    stHomeAdsGroup:= stHomeADS, 
	    bResult_HomeDone=>stAxis.State.bHome_OK, 
	    bResult_HomeBusy=> stAxis.State.bHoming, 
	    bResult_HomeError=>(*stAxis.State.arErrorID[10]*), 
	    nResult_HomeErrorID=> , 
	    axis:=AxisRef );
END_CASE
bHomeExe:=stAxis.Control.bHome_A AND (uiMotionCMD = 3) AND (NOT stAxis.Parameter.bAbsEnc);
bHoming:=stAxis.State.bHoming;
END_IF
END_ACTION

ACTION A_07_Jog:
{region "轴JOG"}
//JOG运动
IF uiMotionCMD = 2 THEN
	bJogFExe:=((stSystem.bManual AND stAxis.Control.bJogCw_M) OR stAxis.control.bJogCw_A) AND stAxis.Control.bJogCw_Con   ;
	bJogBExe :=((stSystem.bManual AND stAxis.Control.bJogCcw_M) OR stAxis.Control.bJogCcw_A) AND stAxis.Control.bJogCcw_Con   ;
	CASE stAxis.Control.iJogMode OF
		0:
			mcJogContinuous(
				Axis:=AxisRef , 
				JogForward:=bJogFExe  AND ( stAxis.Parameter.rJogVel_A<>REAL#0) AND bMoveBaseCon AND NOT fbMcStop.Busy AND NOT bStopMoveExe, 
				JogBackwards:=bJogBExe  AND ( stAxis.Parameter.rJogVel_A<>REAL#0) AND bMoveBaseCon AND NOT fbMcStop.Busy AND NOT bStopMoveExe, 
				Mode:= E_JOGMODE.MC_JOGMODE_CONTINOUS, 
				Position:= , 
				Velocity:= stAxis.Parameter.rJogVel_A  , 
				Acceleration:=stAxis.Parameter.rJogAcc_A, 
				Deceleration:=stAxis.Parameter.rJogDec_A, 
				Jerk:=REAL#100 * stAxis.Parameter.rJogVel_A , 
				Done=> , 
				Busy=> , 
				Active=> , 
				CommandAborted=> , 
				Error=> , 
				ErrorID=> );
		1:
			McJogInching(
				Axis:=AxisRef, 
				JogForward:= bJogFExe AND NOT stAxis.State.bPSw AND ( stAxis.Parameter.rJogVel_A<>REAL#0) AND bMoveBaseCon AND NOT fbMcStop.Busy, 
				JogBackwards:= bJogBExe AND NOT stAxis.State.bNSw AND ( stAxis.Parameter.rJogVel_A<>REAL#0) AND bMoveBaseCon AND NOT fbMcStop.Busy, 
				Mode:= E_JOGMODE.MC_JOGMODE_INCHING, 
				Position:=  stAxis.Parameter.rJogPos_A, 
				Velocity:= stAxis.Parameter.rJogVel_A, 
				Acceleration:=stAxis.Parameter.rJogAcc_A , 
				Deceleration:=stAxis.Parameter.rJogDec_A , 
				Jerk:=REAL#100 * stAxis.Parameter.rJogVel_A , 
				Done=> , 
				Busy=> , 
				Active=> , 
				CommandAborted=> , 
				Error=> , 
				ErrorID=> );
	END_CASE;
END_IF;
{endregion}
END_ACTION

ACTION A_08_Move:

{region "轴定位"}
//定位运动
IF uiMotionCMD = 1 THEN
	bPosUpdate:=FALSE;
	bRelMoveCon:=bMoveBaseCon (*AND NOT AxisRef.Status.Stopping  *);
	bAbsMoveCon:=bMoveBaseCon AND stAxis.State.bHome_OK (*AND NOT AxisRef.Status.Stopping *);
	
	//判断当前是否有新的定位触发
	IF NOT stAxis.Pos.Par.bRelEnable AND (ABS(stAxis.Pos.Par.rPos - stAxis.State.rActPos )<= stAxis.Parameter.rInPosValue)  THEN
		stAxis.Pos.State.bGo_Moving := FALSE ;
		bGO_OK:= TRUE ;
	ELSE			 
		bPosCmd:=((stAxis.Pos.Ctrl.bGo_M AND stSystem.bManual) OR stAxis.Pos.Ctrl.bGo_A) AND NOT AxisRef.Status.Stopping ;
	END_IF;		
	//新的定位命令触发并满足运动条件时，更新目标位置
	IF bPosCmd THEN                                                                       
		IF stAxis.Pos.Ctrl.bGo_Con AND ((stAxis.Pos.Par.bRelEnable AND bRelMoveCon) OR (NOT stAxis.Pos.Par.bRelEnable AND bAbsMoveCon)) 	THEN
			iPosId := 1 ;
			bPosUpdate:=TRUE;
		ELSE
	//轴报警11-定位运动条件不满足报警
			stAxis.State.bLightEror:=TRUE;
			stAxis.State.arErrorID[11]:=TRUE;
		END_IF;
	END_IF;
	//轴报警12-位运动条件不满足报警
	//定位过程中条件不满足报警
	IF stAxis.Pos.State.bGo_Moving THEN
		IF NOT stAxis.Pos.Ctrl.bGo_Con  THEN									
			stAxis.State.bLightEror:=TRUE;
			stAxis.State.arErrorID[12]:=TRUE;
		END_IF;
	END_IF;
		
	//命令复位
	stAxis.Pos.Ctrl.bGo_M:=FALSE;     																		
	stAxis.Pos.Ctrl.bGo_A:=FALSE; 
	
	//命令触发   
	//运动过程中，当前定位参数和目前定位参数不一致，需要重新定位     
	IF iPosId <> -1 THEN                                                                               	
		IF (rVelEx <> stAxis.Pos.Par.rVel) 
			OR (NOT stAxis.Pos.Par.bRelEnable AND (rPosEx <> stAxis.Pos.Par.rPos))
			(* OR (bRelEx <> stAxis.Pos.Par.bRelEnable)*) THEN
				 
			bPosUpdate:=TRUE;
				 
		END_IF;
		IF bPosUpdate THEN
			//复位定位状态                                                          	
			stAxis.Pos.State.bGo_Moving := FALSE;	
			
			//更新当前定位参数
			rRelStartPos := stAxis.State.rActPos;				
			rPosEx:=stAxis.Pos.Par.rPos;                                                              			 
			rVelEx:=stAxis.Pos.Par.rVel;
			rAccEx:=stAxis.Pos.Par.rAcc;
			rDecEx:=stAxis.Pos.Par.rDec;
			rJerkEx:=stAxis.Pos.Par.rJerk;
			bRelEx:=stAxis.Pos.Par.bRelEnable;	
			rVelExTmp := rVelEx;
			
			//触发定位标志														
			IF bRelEx THEN                                                                                       
				bMoveAbsExe:=FALSE;
				bMoveRelExe:=TRUE;					
			ELSE
				bMoveAbsExe:=TRUE;
				bMoveRelExe:=FALSE;					
			END_IF;	
				
			//更新定位指令1编号
			IF	iPosInstNum = 0 THEN																		
				iPosInstNum := 1;
			ELSIF iPosInstNum = 1 THEN
				iPosInstNum := 2;
			ELSIF iPosInstNum = 2 THEN
				iPosInstNum := 1;
			END_IF;			
		END_IF;
	END_IF;

	
//线性轴绝对定位	
	IF  NOT bRelEx THEN																		
		fbMC_MoveA(
			Axis:= AxisRef, 
			Execute:= bMoveAbsExe AND (iPosInstNum = 1), 
			Position:= rPosEx, 
			Velocity:= rVelExTmp, 
			Acceleration:= rAccEx, 
			Deceleration:= rDecEx, 
			Jerk:= rJerkEx, 
			BufferMode:= MC_Aborting, 
			Options:= ,
			Done=> bPosDone1,
			Busy=> bPosBusy1);		
		fbMC_MoveA2(
			Axis:= AxisRef, 
			Execute:= bMoveAbsExe AND (iPosInstNum = 2), 
			Position:= rPosEx, 
			Velocity:= rVelExTmp, 
			Acceleration:= rAccEx, 
			Deceleration:= rDecEx, 
			Jerk:= rJerkEx, 
			BufferMode:= MC_Aborting, 
			Options:= ,
			Done=> bPosDone2,
			Busy=> bPosBusy2);		
			
//线性轴相对定位
	ELSIF  bRelEx THEN										
		fbMC_MoveR(
			Axis:= AxisRef,
			Execute:= bMoveRelExe AND (iPosInstNum = 1), 
			Distance:= rPosEx, 
			Velocity:= rVelExTmp, 
			Acceleration:= rAccEx, 
			Deceleration:= rDecEx, 
			Jerk:= rJerkEx, 
			BufferMode:= MC_Aborting, 
			Options:= ,
			Done=> bPosDone1,
			Busy=> bPosBusy1);	
		fbMC_MoveR2(
			Axis:= AxisRef, 
			Execute:= bMoveRelExe AND (iPosInstNum = 2), 
			Distance:= rPosEx, 
			Velocity:= rVelExTmp, 
			Acceleration:= rAccEx, 
			Deceleration:= rDecEx, 
			Jerk:= rJerkEx, 
			BufferMode:= MC_Aborting, 
			Options:= ,
			Done=> bPosDone2,
			Busy=> bPosBusy2);							 
	END_IF

	bMoveAbsExe:=FALSE;
	bMoveRelExe:=FALSE;		
 
		 
